LIN {X 0,Y 353.763,Z 539.719,A -85,B 0,C 180,E1 -13406.585,E2 -13406.585} C_VEL
LIN {X 0,Y 353.878,Z 540.945,A -85,B 0,C 180,E1 -13408.863,E2 -13408.863} C_VEL
LIN {X 0,Y 353.87,Z 540.944,A -85,B 0,C 180,E1 -13411.139,E2 -13411.139} C_VEL
LIN {X 0,Y 353.763,Z 539.714,A -85,B 0,C 180,E1 -13413.418,E2 -13413.418} C_VEL
LIN {X 0,Y 353.653,Z 537.275,A -85,B 0,C 180,E1 -13415.704,E2 -13415.704} C_VEL
LIN {X 0,Y 353.599,Z 534.658,A -85,B 0,C 180,E1 -13417.424,E2 -13417.424} C_VEL
LIN {X 0,Y 353.603,Z 529.946,A -85,B 0,C 180,E1 -13419.728,E2 -13419.728} C_VEL
LIN {X 0,Y 353.94,Z 523.835,A -85,B 0,C 180,E1 -13422.035,E2 -13422.035} C_VEL
LIN {X 0,Y 354.657,Z 516.159,A -85,B 0,C 180,E1 -13424.343,E2 -13424.343} C_VEL
LIN {X 0,Y 355.631,Z 507.936,A -85,B 0,C 180,E1 -13426.358,E2 -13426.358} C_VEL
LIN {X 0,Y 357.037,Z 498.093,A -85,B 0,C 180,E1 -13428.359,E2 -13428.359} C_VEL
LIN {X 0,Y 358.396,Z 488.39,A -85,B 0,C 180,E1 -13430.012,E2 -13430.012} C_VEL
LIN {X 0,Y 360.06,Z 477.162,A -85,B 0,C 180,E1 -13431.62,E2 -13431.62} C_VEL
LIN {X 0,Y 362.009,Z 464.197,A -85,B 0,C 180,E1 -13433.151,E2 -13433.151} C_VEL
LIN {X 0,Y 363.932,Z 451.379,A -85,B 0,C 180,E1 -13434.381,E2 -13434.381} C_VEL
LIN {X 0,Y 365.533,Z 438.976,A -85,B 0,C 180,E1 -13435.357,E2 -13435.357} C_VEL
LIN {X 0,Y 367.058,Z 425.471,A -85,B 0,C 180,E1 -13436.206,E2 -13436.206} C_VEL
LIN {X 0,Y 368.534,Z 409.817,A -85,B 0,C 180,E1 -13436.932,E2 -13436.932} C_VEL
LIN {X 0,Y 370.623,Z 388.777,A -85,B 0,C 180,E1 -13437.8,E2 -13437.8} C_VEL
LIN {X 0,Y 376.251,Z 305.9,A -85,B 0,C 180,E1 -13440.211,E2 -13440.211} C_VEL
LIN {X 0,Y 378.725,Z 273.446,A -85,B 0,C 180,E1 -13441.214,E2 -13441.214} C_VEL
LIN {X 0,Y 378.077,Z 256.965,A -85,B 0,C 180,E1 -13442.054,E2 -13442.054} C_VEL
LIN {X 0,Y 376.586,Z 241.39,A -85,B 0,C 180,E1 -13443.049,E2 -13443.049} C_VEL
LIN {X 0,Y 375.207,Z 230.072,A -85,B 0,C 180,E1 -13443.907,E2 -13443.907} C_VEL
LIN {X 0,Y 378.638,Z 218.88,A -85,B 0,C 180,E1 -13445.782,E2 -13445.782} C_VEL
LIN {X 0,Y 378.745,Z 217.493,A -85,B 0,C 180,E1 -13446.098,E2 -13446.098} C_VEL
LIN {X 0,Y 377.491,Z 211.701,A -85,B 0,C 180,E1 -13447.908,E2 -13447.908} C_VEL
LIN {X 0,Y 376.04,Z 206.391,A -85,B 0,C 180,E1 -13449.98,E2 -13449.98} C_VEL
LIN {X 0,Y 375.126,Z 203.374,A -85,B 0,C 180,E1 -13451.462,E2 -13451.462} C_VEL
LIN {X 0,Y 374.284,Z 201.061,A -85,B 0,C 180,E1 -13452.92,E2 -13452.92} C_VEL
LIN {X 0,Y 373.576,Z 199.328,A -85,B 0,C 180,E1 -13454.366,E2 -13454.366} C_VEL
LIN {X 0,Y 373.021,Z 198.122,A -85,B 0,C 180,E1 -13455.805,E2 -13455.805} C_VEL
LIN {X 0,Y 372.593,Z 197.372,A -85,B 0,C 180,E1 -13457.362,E2 -13457.362} C_VEL
LIN {X 0,Y 372.29,Z 197.213,A -85,B 0,C 180,E1 -13459.036,E2 -13459.036} C_VEL
LIN {X 0,Y 372.212,Z 198.099,A -85,B 0,C 180,E1 -13461.457,E2 -13461.457} C_VEL
LIN {X 0,Y 372.419,Z 199.091,A -85,B 0,C 180,E1 -13462.852,E2 -13462.852} C_VEL
LIN {X 0,Y 372.909,Z 202.358,A -85,B 0,C 180,E1 -13465.571,E2 -13465.571} C_VEL
LIN {X 0,Y 373.514,Z 206.249,A -85,B 0,C 180,E1 -13467.858,E2 -13467.858} C_VEL
LIN {X 0,Y 374.131,Z 211.79,A -85,B 0,C 180,E1 -13470.359,E2 -13470.359} C_VEL
LIN {X 0,Y 374.358,Z 214.356,A -85,B 0,C 180,E1 -13471.322,E2 -13471.322} C_VEL
LIN {X 0,Y 376.048,Z 218.405,A -85,B 0,C 180,E1 -13471.947,E2 -13471.947} C_VEL
LIN {X 0,Y 379.156,Z 231.614,A -85,B 0,C 180,E1 -13473.357,E2 -13473.357} C_VEL
LIN {X 0,Y 380.829,Z 240.437,A -85,B 0,C 180,E1 -13474.153,E2 -13474.153} C_VEL
LIN {X 0,Y 372.344,Z 323.117,A -85,B 0,C 180,E1 -13477.236,E2 -13477.236} C_VEL
LIN {X 0,Y 371.105,Z 340.845,A -85,B 0,C 180,E1 -13478.009,E2 -13478.009} C_VEL
LIN {X 0,Y 369.933,Z 354.657,A -85,B 0,C 180,E1 -13478.841,E2 -13478.841} C_VEL
LIN {X 0,Y 368.398,Z 368.573,A -85,B 0,C 180,E1 -13479.917,E2 -13479.917} C_VEL
LIN {X 0,Y 366.812,Z 380.901,A -85,B 0,C 180,E1 -13481.136,E2 -13481.136} C_VEL
LIN {X 0,Y 365.241,Z 392.111,A -85,B 0,C 180,E1 -13482.503,E2 -13482.503} C_VEL
LIN {X 0,Y 363.873,Z 400.494,A -85,B 0,C 180,E1 -13483.736,E2 -13483.736} C_VEL
LIN {X 0,Y 362.309,Z 409.709,A -85,B 0,C 180,E1 -13485.394,E2 -13485.394} C_VEL
LIN {X 0,Y 360.749,Z 417.376,A -85,B 0,C 180,E1 -13487.079,E2 -13487.079} C_VEL
LIN {X 0,Y 359.531,Z 423.347,A -85,B 0,C 180,E1 -13488.728,E2 -13488.728} C_VEL
LIN {X 0,Y 358.425,Z 428.175,A -85,B 0,C 180,E1 -13490.406,E2 -13490.406} C_VEL
LIN {X 0,Y 357.393,Z 431.88,A -85,B 0,C 180,E1 -13492.088,E2 -13492.088} C_VEL
LIN {X 0,Y 356.884,Z 433.766,A -85,B 0,C 180,E1 -13493.214,E2 -13493.214} C_VEL
LIN {X 0,Y 356.482,Z 435.152,A -85,B 0,C 180,E1 -13494.343,E2 -13494.343} C_VEL
LIN {X 0,Y 356.177,Z 436.114,A -85,B 0,C 180,E1 -13495.473,E2 -13495.473} C_VEL
LIN {X 0,Y 355.831,Z 436.688,A -85,B 0,C 180,E1 -13496.603,E2 -13496.603} C_VEL
LIN {X 0,Y 355.599,Z 436.836,A -85,B 0,C 180,E1 -13497.735,E2 -13497.735} C_VEL
LIN {X 0,Y 355.294,Z 436.541,A -85,B 0,C 180,E1 -13498.867,E2 -13498.867} C_VEL
LIN {X 0,Y 355.053,Z 435.824,A -85,B 0,C 180,E1 -13500,E2 -13500} C_VEL
LIN {X 0,Y 355.066,Z 434.672,A -85,B 0,C 180,E1 -13501.134,E2 -13501.134} C_VEL
LIN {X 0,Y 354.989,Z 432.145,A -85,B 0,C 180,E1 -13502.837,E2 -13502.837} C_VEL
LIN {X 0,Y 354.872,Z 428.61,A -85,B 0,C 180,E1 -13504.544,E2 -13504.544} C_VEL
LIN {X 0,Y 355.241,Z 423.954,A -85,B 0,C 180,E1 -13506.247,E2 -13506.247} C_VEL
LIN {X 0,Y 355.504,Z 418.114,A -85,B 0,C 180,E1 -13507.954,E2 -13507.954} C_VEL
LIN {X 0,Y 355.863,Z 410.905,A -85,B 0,C 180,E1 -13509.664,E2 -13509.664} C_VEL
LIN {X 0,Y 356.433,Z 402.004,A -85,B 0,C 180,E1 -13511.372,E2 -13511.372} C_VEL
LIN {X 0,Y 357.108,Z 391.08,A -85,B 0,C 180,E1 -13513.081,E2 -13513.081} C_VEL
LIN {X 0,Y 357.776,Z 379.778,A -85,B 0,C 180,E1 -13514.505,E2 -13514.505} C_VEL
LIN {X 0,Y 358.472,Z 367.292,A -85,B 0,C 180,E1 -13515.785,E2 -13515.785} C_VEL
LIN {X 0,Y 359.034,Z 354.854,A -85,B 0,C 180,E1 -13516.803,E2 -13516.803} C_VEL
LIN {X 0,Y 359.607,Z 340.6,A -85,B 0,C 180,E1 -13517.707,E2 -13517.707} C_VEL
LIN {X 0,Y 359.969,Z 327.731,A -85,B 0,C 180,E1 -13518.313,E2 -13518.313} C_VEL
LIN {X 0,Y 360.423,Z 308.207,A -85,B 0,C 180,E1 -13518.916,E2 -13518.916} C_VEL
LIN {X 0,Y 362.911,Z 226.278,A -85,B 0,C 180,E1 -13521.162,E2 -13521.162} C_VEL
LIN {X 0,Y 359.275,Z 202.978,A -85,B 0,C 180,E1 -13522.026,E2 -13522.026} C_VEL
LIN {X 0,Y 360.736,Z 186.431,A -85,B 0,C 180,E1 -13525.38,E2 -13525.38} C_VEL
LIN {X 0,Y 360.386,Z 182.557,A -85,B 0,C 180,E1 -13526.224,E2 -13526.224} C_VEL
LIN {X 0,Y 357.643,Z 170.027,A -85,B 0,C 180,E1 -13529.101,E2 -13529.101} C_VEL
LIN {X 0,Y 354.837,Z 157.912,A -85,B 0,C 180,E1 -13532.024,E2 -13532.024} C_VEL
LIN {X 0,Y 354.827,Z 157.912,A -85,B 0,C 180,E1 -13535.699,E2 -13535.699} C_VEL
LIN {X 0,Y 354.804,Z 157.904,A -85,B 0,C 180,E1 -13539.418,E2 -13539.418} C_VEL
LIN {X 0,Y 354.791,Z 157.912,A -85,B 0,C 180,E1 -13542.866,E2 -13542.866} C_VEL
LIN {X 0,Y 354.786,Z 157.915,A -85,B 0,C 180,E1 -13546.105,E2 -13546.105} C_VEL
LIN {X 0,Y 354.793,Z 157.914,A -85,B 0,C 180,E1 -13549.178,E2 -13549.178} C_VEL
LIN {X 0,Y 354.812,Z 157.912,A -85,B 0,C 180,E1 -13552.402,E2 -13552.402} C_VEL
LIN {X 0,Y 354.888,Z 158.025,A -85,B 0,C 180,E1 -13555.059,E2 -13555.059} C_VEL
LIN {X 0,Y 359.7,Z 171.926,A -85,B 0,C 180,E1 -13557.692,E2 -13557.692} C_VEL
LIN {X 0,Y 369.684,Z 191.582,A -85,B 0,C 180,E1 -13559.124,E2 -13559.124} C_VEL
LIN {X 0,Y 374.764,Z 202.976,A -85,B 0,C 180,E1 -13559.846,E2 -13559.846} C_VEL
LIN {X 0,Y 372.675,Z 285.003,A -85,B 0,C 180,E1 -13561.448,E2 -13561.448} C_VEL
LIN {X 0,Y 371.249,Z 338.669,A -85,B 0,C 180,E1 -13562.519,E2 -13562.519} C_VEL
LIN {X 0,Y 370.646,Z 353.596,A -85,B 0,C 180,E1 -13563.016,E2 -13563.016} C_VEL
LIN {X 0,Y 369.847,Z 366.135,A -85,B 0,C 180,E1 -13563.599,E2 -13563.599} C_VEL
LIN {X 0,Y 368.737,Z 380.111,A -85,B 0,C 180,E1 -13564.453,E2 -13564.453} C_VEL
LIN {X 0,Y 367.253,Z 394.224,A -85,B 0,C 180,E1 -13565.553,E2 -13565.553} C_VEL
LIN {X 0,Y 365.586,Z 407.061,A -85,B 0,C 180,E1 -13566.789,E2 -13566.789} C_VEL
LIN {X 0,Y 363.719,Z 419.822,A -85,B 0,C 180,E1 -13568.297,E2 -13568.297} C_VEL
LIN {X 0,Y 362.183,Z 430.662,A -85,B 0,C 180,E1 -13569.852,E2 -13569.852} C_VEL
LIN {X 0,Y 360.499,Z 440.551,A -85,B 0,C 180,E1 -13571.529,E2 -13571.529} C_VEL
LIN {X 0,Y 358.745,Z 450.446,A -85,B 0,C 180,E1 -13573.554,E2 -13573.554} C_VEL
LIN {X 0,Y 357.303,Z 459.202,A -85,B 0,C 180,E1 -13575.765,E2 -13575.765} C_VEL
LIN {X 0,Y 356.039,Z 466.459,A -85,B 0,C 180,E1 -13578.037,E2 -13578.037} C_VEL
LIN {X 0,Y 355.175,Z 472.199,A -85,B 0,C 180,E1 -13580.316,E2 -13580.316} C_VEL
LIN {X 0,Y 354.597,Z 476.084,A -85,B 0,C 180,E1 -13582.302,E2 -13582.302} C_VEL
LIN {X 0,Y 354.189,Z 479.036,A -85,B 0,C 180,E1 -13584.305,E2 -13584.305} C_VEL
LIN {X 0,Y 353.991,Z 481.303,A -85,B 0,C 180,E1 -13586.584,E2 -13586.584} C_VEL
LIN {X 0,Y 353.777,Z 482.464,A -85,B 0,C 180,E1 -13588.86,E2 -13588.86} C_VEL
LIN {X 0,Y 353.777,Z 482.478,A -85,B 0,C 180,E1 -13591.137,E2 -13591.137} C_VEL
LIN {X 0,Y 353.85,Z 482.051,A -85,B 0,C 180,E1 -13592.295,E2 -13592.295} C_VEL
LIN {X 0,Y 353.242,Z 481.561,A -85,B 0,C 180,E1 -13593.242,E2 -13593.242} C_VEL
LIN {X 0,Y 350.492,Z 480.531,A -85,B 0,C 180,E1 -13594.786,E2 -13594.786} C_VEL
LIN {X 0,Y 348.245,Z 479.373,A -85,B 0,C 180,E1 -13596.027,E2 -13596.027} C_VEL
LIN {X 0,Y 347.422,Z 478.194,A -85,B 0,C 180,E1 -13596.975,E2 -13596.975} C_VEL
LIN {X 0,Y 347.431,Z 477.716,A -85,B 0,C 180,E1 -13597.292,E2 -13597.292} C_VEL
LIN {X 0,Y 347.976,Z 474.204,A -85,B 0,C 180,E1 -13599.297,E2 -13599.297} C_VEL
LIN {X 0,Y 348.813,Z 468.885,A -85,B 0,C 180,E1 -13601.622,E2 -13601.622} C_VEL
LIN {X 0,Y 349.961,Z 462.092,A -85,B 0,C 180,E1 -13603.943,E2 -13603.943} C_VEL
LIN {X 0,Y 351.287,Z 454.677,A -85,B 0,C 180,E1 -13605.997,E2 -13605.997} C_VEL
LIN {X 0,Y 352.908,Z 445.996,A -85,B 0,C 180,E1 -13607.978,E2 -13607.978} C_VEL
LIN {X 0,Y 354.83,Z 435.328,A -85,B 0,C 180,E1 -13609.977,E2 -13609.977} C_VEL
LIN {X 0,Y 356.6,Z 424.361,A -85,B 0,C 180,E1 -13611.685,E2 -13611.685} C_VEL
LIN {X 0,Y 358.482,Z 412.292,A -85,B 0,C 180,E1 -13613.236,E2 -13613.236} C_VEL
LIN {X 0,Y 360.37,Z 398.941,A -85,B 0,C 180,E1 -13614.635,E2 -13614.635} C_VEL
LIN {X 0,Y 361.89,Z 385.861,A -85,B 0,C 180,E1 -13615.753,E2 -13615.753} C_VEL
LIN {X 0,Y 363.247,Z 372.108,A -85,B 0,C 180,E1 -13616.688,E2 -13616.688} C_VEL
LIN {X 0,Y 364.171,Z 357.951,A -85,B 0,C 180,E1 -13617.438,E2 -13617.438} C_VEL
LIN {X 0,Y 364.941,Z 342.964,A -85,B 0,C 180,E1 -13617.994,E2 -13617.994} C_VEL
LIN {X 0,Y 365.469,Z 322.552,A -85,B 0,C 180,E1 -13618.458,E2 -13618.458} C_VEL
LIN {X 0,Y 368.091,Z 226.756,A -85,B 0,C 180,E1 -13620.348,E2 -13620.348} C_VEL
LIN {X 0,Y 368.573,Z 204.816,A -85,B 0,C 180,E1 -13620.794,E2 -13620.794} C_VEL
LIN {X 0,Y 361.129,Z 188.738,A -85,B 0,C 180,E1 -13621.884,E2 -13621.884} C_VEL
LIN {X 0,Y 352.618,Z 172.366,A -85,B 0,C 180,E1 -13623.165,E2 -13623.165} C_VEL
LIN {X 0,Y 347.762,Z 158.793,A -85,B 0,C 180,E1 -13625.847,E2 -13625.847} C_VEL
LIN {X 0,Y 347.747,Z 158.778,A -85,B 0,C 180,E1 -13628.791,E2 -13628.791} C_VEL
LIN {X 0,Y 347.748,Z 158.783,A -85,B 0,C 180,E1 -13631.828,E2 -13631.828} C_VEL
LIN {X 0,Y 347.727,Z 158.79,A -85,B 0,C 180,E1 -13635.021,E2 -13635.021} C_VEL
LIN {X 0,Y 347.761,Z 158.787,A -85,B 0,C 180,E1 -13638.393,E2 -13638.393} C_VEL
LIN {X 0,Y 347.768,Z 158.785,A -85,B 0,C 180,E1 -13642.009,E2 -13642.009} C_VEL
LIN {X 0,Y 347.736,Z 158.783,A -85,B 0,C 180,E1 -13645.535,E2 -13645.535} C_VEL
LIN {X 0,Y 347.756,Z 158.791,A -85,B 0,C 180,E1 -13648.301,E2 -13648.301} C_VEL
LIN {X 0,Y 347.797,Z 158.775,A -85,B 0,C 180,E1 -13650.989,E2 -13650.989} C_VEL
LIN {X 0,Y 347.822,Z 158.779,A -85,B 0,C 180,E1 -13653.607,E2 -13653.607} C_VEL
LIN {X 0,Y 347.775,Z 158.779,A -85,B 0,C 180,E1 -13656.161,E2 -13656.161} C_VEL
LIN {X 0,Y 347.801,Z 158.776,A -85,B 0,C 180,E1 -13659.909,E2 -13659.909} C_VEL
LIN {X 0,Y 347.856,Z 158.77,A -85,B 0,C 180,E1 -13662.359,E2 -13662.359} C_VEL
LIN {X 0,Y 347.887,Z 158.765,A -85,B 0,C 180,E1 -13665.97,E2 -13665.97} C_VEL
LIN {X 0,Y 347.918,Z 158.771,A -85,B 0,C 180,E1 -13669.525,E2 -13669.525} C_VEL
LIN {X 0,Y 348.063,Z 158.747,A -85,B 0,C 180,E1 -13671.874,E2 -13671.874} C_VEL
LIN {X 0,Y 348.057,Z 158.734,A -85,B 0,C 180,E1 -13674.205,E2 -13674.205} C_VEL
LIN {X 0,Y 348.198,Z 158.734,A -85,B 0,C 180,E1 -13677.686,E2 -13677.686} C_VEL
LIN {X 0,Y 348.358,Z 158.695,A -85,B 0,C 180,E1 -13680,E2 -13680} C_VEL
LIN {X 0,Y 348.198,Z 158.73,A -85,B 0,C 180,E1 -13682.313,E2 -13682.313} C_VEL
LIN {X 0,Y 348.095,Z 158.727,A -85,B 0,C 180,E1 -13686.958,E2 -13686.958} C_VEL
LIN {X 0,Y 347.956,Z 158.762,A -85,B 0,C 180,E1 -13689.299,E2 -13689.299} C_VEL
LIN {X 0,Y 347.879,Z 158.753,A -85,B 0,C 180,E1 -13692.84,E2 -13692.84} C_VEL
LIN {X 0,Y 347.83,Z 158.78,A -85,B 0,C 180,E1 -13696.432,E2 -13696.432} C_VEL
LIN {X 0,Y 347.84,Z 158.761,A -85,B 0,C 180,E1 -13698.861,E2 -13698.861} C_VEL
LIN {X 0,Y 347.764,Z 158.786,A -85,B 0,C 180,E1 -13702.58,E2 -13702.58} C_VEL
LIN {X 0,Y 347.801,Z 158.772,A -85,B 0,C 180,E1 -13705.109,E2 -13705.109} C_VEL
LIN {X 0,Y 347.798,Z 158.786,A -85,B 0,C 180,E1 -13707.695,E2 -13707.695} C_VEL
LIN {X 0,Y 347.739,Z 158.783,A -85,B 0,C 180,E1 -13710.349,E2 -13710.349} C_VEL
LIN {X 0,Y 347.738,Z 158.784,A -85,B 0,C 180,E1 -13714.045,E2 -13714.045} C_VEL
LIN {X 0,Y 347.757,Z 158.79,A -85,B 0,C 180,E1 -13717.321,E2 -13717.321} C_VEL
LIN {X 0,Y 347.722,Z 158.752,A -85,B 0,C 180,E1 -13720.298,E2 -13720.298} C_VEL
LIN {X 0,Y 347.72,Z 158.795,A -85,B 0,C 180,E1 -13723.408,E2 -13723.408} C_VEL
LIN {X 0,Y 347.778,Z 158.79,A -85,B 0,C 180,E1 -13726.677,E2 -13726.677} C_VEL
LIN {X 0,Y 347.827,Z 158.983,A -85,B 0,C 180,E1 -13728.726,E2 -13728.726} C_VEL
LIN {X 0,Y 353.697,Z 178.827,A -85,B 0,C 180,E1 -13732.395,E2 -13732.395} C_VEL
LIN {X 0,Y 359.113,Z 197.549,A -85,B 0,C 180,E1 -13735.625,E2 -13735.625} C_VEL
LIN {X 0,Y 360.254,Z 202.214,A -85,B 0,C 180,E1 -13736.391,E2 -13736.391} C_VEL
LIN {X 0,Y 359.364,Z 209.237,A -85,B 0,C 180,E1 -13737.323,E2 -13737.323} C_VEL
LIN {X 0,Y 360.134,Z 219.316,A -85,B 0,C 180,E1 -13737.839,E2 -13737.839} C_VEL
LIN {X 0,Y 365.985,Z 269.667,A -85,B 0,C 180,E1 -13739.525,E2 -13739.525} C_VEL
LIN {X 0,Y 366.395,Z 275.472,A -85,B 0,C 180,E1 -13739.69,E2 -13739.69} C_VEL
LIN {X 0,Y 363.207,Z 392.946,A -85,B 0,C 180,E1 -13742.017,E2 -13742.017} C_VEL
LIN {X 0,Y 362.288,Z 407.953,A -85,B 0,C 180,E1 -13742.49,E2 -13742.49} C_VEL
LIN {X 0,Y 360.903,Z 422.665,A -85,B 0,C 180,E1 -13743.159,E2 -13743.159} C_VEL
LIN {X 0,Y 359.199,Z 437.235,A -85,B 0,C 180,E1 -13744.055,E2 -13744.055} C_VEL
LIN {X 0,Y 357.445,Z 451.111,A -85,B 0,C 180,E1 -13745.161,E2 -13745.161} C_VEL
LIN {X 0,Y 355.396,Z 463.777,A -85,B 0,C 180,E1 -13746.396,E2 -13746.396} C_VEL
LIN {X 0,Y 353.42,Z 476.713,A -85,B 0,C 180,E1 -13747.956,E2 -13747.956} C_VEL
LIN {X 0,Y 351.695,Z 487.545,A -85,B 0,C 180,E1 -13749.532,E2 -13749.532} C_VEL
LIN {X 0,Y 350.176,Z 497.585,A -85,B 0,C 180,E1 -13751.271,E2 -13751.271} C_VEL
LIN {X 0,Y 348.867,Z 506.148,A -85,B 0,C 180,E1 -13753.018,E2 -13753.018} C_VEL
LIN {X 0,Y 347.793,Z 514.543,A -85,B 0,C 180,E1 -13755.071,E2 -13755.071} C_VEL
LIN {X 0,Y 347.028,Z 521.509,A -85,B 0,C 180,E1 -13757.13,E2 -13757.13} C_VEL
LIN {X 0,Y 346.539,Z 527.985,A -85,B 0,C 180,E1 -13759.485,E2 -13759.485} C_VEL
LIN {X 0,Y 346.461,Z 533.011,A -85,B 0,C 180,E1 -13761.838,E2 -13761.838} C_VEL
LIN {X 0,Y 346.563,Z 536.701,A -85,B 0,C 180,E1 -13764.182,E2 -13764.182} C_VEL
LIN {X 0,Y 346.665,Z 539.132,A -85,B 0,C 180,E1 -13766.515,E2 -13766.515} C_VEL
LIN {X 0,Y 346.824,Z 540.362,A -85,B 0,C 180,E1 -13768.84,E2 -13768.84} C_VEL
LIN {X 0,Y 346.817,Z 540.361,A -85,B 0,C 180,E1 -13771.163,E2 -13771.163} C_VEL
LIN {X 0,Y 346.665,Z 539.126,A -85,B 0,C 180,E1 -13773.488,E2 -13773.488} C_VEL
LIN {X 0,Y 346.582,Z 536.688,A -85,B 0,C 180,E1 -13775.821,E2 -13775.821} C_VEL
LIN {X 0,Y 346.479,Z 532.983,A -85,B 0,C 180,E1 -13778.164,E2 -13778.164} C_VEL
LIN {X 0,Y 346.578,Z 527.946,A -85,B 0,C 180,E1 -13780.517,E2 -13780.517} C_VEL
LIN {X 0,Y 347.068,Z 521.466,A -85,B 0,C 180,E1 -13782.872,E2 -13782.872} C_VEL
LIN {X 0,Y 347.81,Z 514.488,A -85,B 0,C 180,E1 -13784.931,E2 -13784.931} C_VEL
LIN {X 0,Y 348.919,Z 506.079,A -85,B 0,C 180,E1 -13786.983,E2 -13786.983} C_VEL
LIN {X 0,Y 350.429,Z 496.148,A -85,B 0,C 180,E1 -13788.988,E2 -13788.988} C_VEL
LIN {X 0,Y 351.991,Z 485.637,A -85,B 0,C 180,E1 -13790.758,E2 -13790.758} C_VEL
LIN {X 0,Y 353.965,Z 473.341,A -85,B 0,C 180,E1 -13792.472,E2 -13792.472} C_VEL
LIN {X 0,Y 356.088,Z 459.655,A -85,B 0,C 180,E1 -13794.022,E2 -13794.022} C_VEL
LIN {X 0,Y 358.062,Z 445.95,A -85,B 0,C 180,E1 -13795.273,E2 -13795.273} C_VEL
LIN {X 0,Y 359.886,Z 431.721,A -85,B 0,C 180,E1 -13796.3,E2 -13796.3} C_VEL
LIN {X 0,Y 361.501,Z 417.029,A -85,B 0,C 180,E1 -13797.108,E2 -13797.108} C_VEL
LIN {X 0,Y 363.932,Z 398.14,A -85,B 0,C 180,E1 -13798.082,E2 -13798.082} C_VEL
LIN {X 0,Y 365.464,Z 381.659,A -85,B 0,C 180,E1 -13798.697,E2 -13798.697} C_VEL
LIN {X 0,Y 370.169,Z 317.229,A -85,B 0,C 180,E1 -13800.603,E2 -13800.603} C_VEL
LIN {X 0,Y 373.714,Z 274.991,A -85,B 0,C 180,E1 -13801.938,E2 -13801.938} C_VEL
LIN {X 0,Y 373.221,Z 259.069,A -85,B 0,C 180,E1 -13802.777,E2 -13802.777} C_VEL
LIN {X 0,Y 371.973,Z 243.743,A -85,B 0,C 180,E1 -13803.791,E2 -13803.791} C_VEL
LIN {X 0,Y 370.399,Z 229.425,A -85,B 0,C 180,E1 -13804.945,E2 -13804.945} C_VEL
LIN {X 0,Y 373.015,Z 221.289,A -85,B 0,C 180,E1 -13806.381,E2 -13806.381} C_VEL
LIN {X 0,Y 371.827,Z 215.544,A -85,B 0,C 180,E1 -13808.241,E2 -13808.241} C_VEL
LIN {X 0,Y 370.359,Z 209.828,A -85,B 0,C 180,E1 -13810.62,E2 -13810.62} C_VEL
LIN {X 0,Y 369.48,Z 207.102,A -85,B 0,C 180,E1 -13812.112,E2 -13812.112} C_VEL
LIN {X 0,Y 368.695,Z 205.03,A -85,B 0,C 180,E1 -13813.585,E2 -13813.585} C_VEL
LIN {X 0,Y 368.052,Z 203.519,A -85,B 0,C 180,E1 -13815.048,E2 -13815.048} C_VEL
LIN {X 0,Y 367.52,Z 202.469,A -85,B 0,C 180,E1 -13816.609,E2 -13816.609} C_VEL
LIN {X 0,Y 367.155,Z 201.985,A -85,B 0,C 180,E1 -13818.292,E2 -13818.292} C_VEL
LIN {X 0,Y 366.898,Z 202.44,A -85,B 0,C 180,E1 -13820.793,E2 -13820.793} C_VEL
LIN {X 0,Y 366.958,Z 203.261,A -85,B 0,C 180,E1 -13822.203,E2 -13822.203} C_VEL
LIN {X 0,Y 367.3,Z 206.132,A -85,B 0,C 180,E1 -13824.969,E2 -13824.969} C_VEL
LIN {X 0,Y 367.772,Z 209.601,A -85,B 0,C 180,E1 -13827.229,E2 -13827.229} C_VEL
LIN {X 0,Y 368.272,Z 214.827,A -85,B 0,C 180,E1 -13829.773,E2 -13829.773} C_VEL
LIN {X 0,Y 368.538,Z 215.694,A -85,B 0,C 180,E1 -13830.04,E2 -13830.04} C_VEL
LIN {X 0,Y 371.209,Z 220.927,A -85,B 0,C 180,E1 -13831.065,E2 -13831.065} C_VEL
LIN {X 0,Y 372.143,Z 223.669,A -85,B 0,C 180,E1 -13831.464,E2 -13831.464} C_VEL
LIN {X 0,Y 374.899,Z 236.499,A -85,B 0,C 180,E1 -13832.858,E2 -13832.858} C_VEL
LIN {X 0,Y 375.941,Z 242.696,A -85,B 0,C 180,E1 -13833.428,E2 -13833.428} C_VEL
LIN {X 0,Y 366.955,Z 323.86,A -85,B 0,C 180,E1 -13836.532,E2 -13836.532} C_VEL
LIN {X 0,Y 365.598,Z 341.651,A -85,B 0,C 180,E1 -13837.329,E2 -13837.329} C_VEL
LIN {X 0,Y 364.363,Z 354.916,A -85,B 0,C 180,E1 -13838.134,E2 -13838.134} C_VEL
LIN {X 0,Y 362.669,Z 369.199,A -85,B 0,C 180,E1 -13839.252,E2 -13839.252} C_VEL
LIN {X 0,Y 360.919,Z 381.86,A -85,B 0,C 180,E1 -13840.521,E2 -13840.521} C_VEL
LIN {X 0,Y 359.214,Z 393.033,A -85,B 0,C 180,E1 -13841.905,E2 -13841.905} C_VEL
LIN {X 0,Y 357.737,Z 401.41,A -85,B 0,C 180,E1 -13843.156,E2 -13843.156} C_VEL
LIN {X 0,Y 356.051,Z 410.649,A -85,B 0,C 180,E1 -13844.839,E2 -13844.839} C_VEL
LIN {X 0,Y 354.316,Z 418.652,A -85,B 0,C 180,E1 -13846.632,E2 -13846.632} C_VEL
LIN {X 0,Y 352.819,Z 425.248,A -85,B 0,C 180,E1 -13848.51,E2 -13848.51} C_VEL
LIN {X 0,Y 351.647,Z 429.9,A -85,B 0,C 180,E1 -13850.219,E2 -13850.219} C_VEL
LIN {X 0,Y 350.561,Z 433.461,A -85,B 0,C 180,E1 -13851.933,E2 -13851.933} C_VEL
LIN {X 0,Y 349.99,Z 435.223,A -85,B 0,C 180,E1 -13853.08,E2 -13853.08} C_VEL
LIN {X 0,Y 349.568,Z 436.525,A -85,B 0,C 180,E1 -13854.231,E2 -13854.231} C_VEL
LIN {X 0,Y 349.221,Z 437.423,A -85,B 0,C 180,E1 -13855.383,E2 -13855.383} C_VEL
LIN {X 0,Y 348.858,Z 437.921,A -85,B 0,C 180,E1 -13856.535,E2 -13856.535} C_VEL
LIN {X 0,Y 348.608,Z 437.957,A -85,B 0,C 180,E1 -13857.689,E2 -13857.689} C_VEL
LIN {X 0,Y 348.285,Z 437.584,A -85,B 0,C 180,E1 -13858.844,E2 -13858.844} C_VEL
LIN {X 0,Y 348.026,Z 436.798,A -85,B 0,C 180,E1 -13860,E2 -13860} C_VEL
LIN {X 0,Y 348.04,Z 435.574,A -85,B 0,C 180,E1 -13861.157,E2 -13861.157} C_VEL
LIN {X 0,Y 347.951,Z 432.916,A -85,B 0,C 180,E1 -13862.895,E2 -13862.895} C_VEL
LIN {X 0,Y 347.844,Z 429.246,A -85,B 0,C 180,E1 -13864.636,E2 -13864.636} C_VEL
LIN {X 0,Y 348.201,Z 424.451,A -85,B 0,C 180,E1 -13866.374,E2 -13866.374} C_VEL
LIN {X 0,Y 348.477,Z 418.463,A -85,B 0,C 180,E1 -13868.116,E2 -13868.116} C_VEL
LIN {X 0,Y 348.85,Z 411.051,A -85,B 0,C 180,E1 -13869.86,E2 -13869.86} C_VEL
LIN {X 0,Y 349.437,Z 401.938,A -85,B 0,C 180,E1 -13871.603,E2 -13871.603} C_VEL
LIN {X 0,Y 350.09,Z 391.773,A -85,B 0,C 180,E1 -13873.2,E2 -13873.2} C_VEL
LIN {X 0,Y 350.778,Z 380.414,A -85,B 0,C 180,E1 -13874.652,E2 -13874.652} C_VEL
LIN {X 0,Y 351.479,Z 367.878,A -85,B 0,C 180,E1 -13875.958,E2 -13875.958} C_VEL
LIN {X 0,Y 352.078,Z 355.174,A -85,B 0,C 180,E1 -13877.011,E2 -13877.011} C_VEL
LIN {X 0,Y 352.657,Z 341.115,A -85,B 0,C 180,E1 -13877.918,E2 -13877.918} C_VEL
LIN {X 0,Y 353.037,Z 328.228,A -85,B 0,C 180,E1 -13878.536,E2 -13878.536} C_VEL
LIN {X 0,Y 353.519,Z 307.596,A -85,B 0,C 180,E1 -13879.187,E2 -13879.187} C_VEL
LIN {X 0,Y 356.105,Z 227.175,A -85,B 0,C 180,E1 -13881.45,E2 -13881.45} C_VEL
LIN {X 0,Y 352.399,Z 203.154,A -85,B 0,C 180,E1 -13882.383,E2 -13882.383} C_VEL
LIN {X 0,Y 353.845,Z 187.528,A -85,B 0,C 180,E1 -13885.594,E2 -13885.594} C_VEL
LIN {X 0,Y 353.382,Z 183.465,A -85,B 0,C 180,E1 -13886.496,E2 -13886.496} C_VEL
LIN {X 0,Y 350.612,Z 171,A -85,B 0,C 180,E1 -13889.413,E2 -13889.413} C_VEL
LIN {X 0,Y 347.772,Z 158.791,A -85,B 0,C 180,E1 -13892.373,E2 -13892.373} C_VEL
LIN {X 0,Y 347.775,Z 158.79,A -85,B 0,C 180,E1 -13896.064,E2 -13896.064} C_VEL
LIN {X 0,Y 347.737,Z 158.79,A -85,B 0,C 180,E1 -13898.795,E2 -13898.795} C_VEL
LIN {X 0,Y 347.753,Z 158.793,A -85,B 0,C 180,E1 -13901.83,E2 -13901.83} C_VEL
LIN {X 0,Y 347.772,Z 158.788,A -85,B 0,C 180,E1 -13905.016,E2 -13905.016} C_VEL
LIN {X 0,Y 347.756,Z 158.793,A -85,B 0,C 180,E1 -13908.396,E2 -13908.396} C_VEL
LIN {X 0,Y 347.778,Z 158.791,A -85,B 0,C 180,E1 -13912.011,E2 -13912.011} C_VEL
LIN {X 0,Y 347.786,Z 158.793,A -85,B 0,C 180,E1 -13914.298,E2 -13914.298} C_VEL
LIN {X 0,Y 352.675,Z 172.62,A -85,B 0,C 180,E1 -13916.97,E2 -13916.97} C_VEL
LIN {X 0,Y 362.527,Z 191.569,A -85,B 0,C 180,E1 -13918.431,E2 -13918.431} C_VEL
LIN {X 0,Y 368.636,Z 204.951,A -85,B 0,C 180,E1 -13919.324,E2 -13919.324} C_VEL
LIN {X 0,Y 366.448,Z 285.768,A -85,B 0,C 180,E1 -13920.923,E2 -13920.923} C_VEL
LIN {X 0,Y 364.942,Z 340.552,A -85,B 0,C 180,E1 -13922.042,E2 -13922.042} C_VEL
LIN {X 0,Y 364.238,Z 355.662,A -85,B 0,C 180,E1 -13922.57,E2 -13922.57} C_VEL
LIN {X 0,Y 363.324,Z 370.003,A -85,B 0,C 180,E1 -13923.294,E2 -13923.294} C_VEL
LIN {X 0,Y 362.204,Z 382.587,A -85,B 0,C 180,E1 -13924.113,E2 -13924.113} C_VEL
LIN {X 0,Y 360.652,Z 396.322,A -85,B 0,C 180,E1 -13925.229,E2 -13925.229} C_VEL
LIN {X 0,Y 358.709,Z 410.137,A -85,B 0,C 180,E1 -13926.624,E2 -13926.624} C_VEL
LIN {X 0,Y 356.808,Z 422.574,A -85,B 0,C 180,E1 -13928.173,E2 -13928.173} C_VEL
LIN {X 0,Y 355.232,Z 432.971,A -85,B 0,C 180,E1 -13929.742,E2 -13929.742} C_VEL
LIN {X 0,Y 353.513,Z 442.593,A -85,B 0,C 180,E1 -13931.451,E2 -13931.451} C_VEL
LIN {X 0,Y 351.962,Z 451.03,A -85,B 0,C 180,E1 -13933.228,E2 -13933.228} C_VEL
LIN {X 0,Y 350.443,Z 459.787,A -85,B 0,C 180,E1 -13935.481,E2 -13935.481} C_VEL
LIN {X 0,Y 349.12,Z 467.044,A -85,B 0,C 180,E1 -13937.796,E2 -13937.796} C_VEL
LIN {X 0,Y 348.187,Z 472.785,A -85,B 0,C 180,E1 -13940.12,E2 -13940.12} C_VEL
LIN {X 0,Y 347.562,Z 476.822,A -85,B 0,C 180,E1 -13942.233,E2 -13942.233} C_VEL
LIN {X 0,Y 347.135,Z 479.622,A -85,B 0,C 180,E1 -13944.189,E2 -13944.189} C_VEL
LIN {X 0,Y 346.938,Z 481.887,A -85,B 0,C 180,E1 -13946.514,E2 -13946.514} C_VEL
LIN {X 0,Y 346.702,Z 483.049,A -85,B 0,C 180,E1 -13948.837,E2 -13948.837} C_VEL
LIN {X 0,Y 346.702,Z 483.063,A -85,B 0,C 180,E1 -13951.16,E2 -13951.16} C_VEL
LIN {X 0,Y 346.935,Z 481.954,A -85,B 0,C 180,E1 -13953.483,E2 -13953.483} C_VEL
LIN {X 0,Y 347.122,Z 479.747,A -85,B 0,C 180,E1 -13955.809,E2 -13955.809} C_VEL
LIN {X 0,Y 347.431,Z 477.716,A -85,B 0,C 180,E1 -13957.292,E2 -13957.292} C_VEL
LIN {X 0,Y 347.046,Z 476.273,A -85,B 0,C 180,E1 -13958.235,E2 -13958.235} C_VEL
LIN {X 0,Y 344.635,Z 473.732,A -85,B 0,C 180,E1 -13959.774,E2 -13959.774} C_VEL
LIN {X 0,Y 342.635,Z 471.38,A -85,B 0,C 180,E1 -13961,E2 -13961} C_VEL
LIN {X 0,Y 341.982,Z 469.302,A -85,B 0,C 180,E1 -13961.923,E2 -13961.923} C_VEL
LIN {X 0,Y 342.045,Z 468.505,A -85,B 0,C 180,E1 -13962.228,E2 -13962.228} C_VEL
LIN {X 0,Y 343.078,Z 462.675,A -85,B 0,C 180,E1 -13964.229,E2 -13964.229} C_VEL
LIN {X 0,Y 344.429,Z 455.517,A -85,B 0,C 180,E1 -13966.258,E2 -13966.258} C_VEL
LIN {X 0,Y 346.189,Z 446.574,A -85,B 0,C 180,E1 -13968.339,E2 -13968.339} C_VEL
LIN {X 0,Y 348.186,Z 435.903,A -85,B 0,C 180,E1 -13970.375,E2 -13970.375} C_VEL
LIN {X 0,Y 350.02,Z 424.936,A -85,B 0,C 180,E1 -13972.114,E2 -13972.114} C_VEL
LIN {X 0,Y 351.982,Z 412.862,A -85,B 0,C 180,E1 -13973.691,E2 -13973.691} C_VEL
LIN {X 0,Y 353.946,Z 399.506,A -85,B 0,C 180,E1 -13975.112,E2 -13975.112} C_VEL
LIN {X 0,Y 355.539,Z 386.417,A -85,B 0,C 180,E1 -13976.248,E2 -13976.248} C_VEL
LIN {X 0,Y 356.931,Z 372.786,A -85,B 0,C 180,E1 -13977.19,E2 -13977.19} C_VEL
LIN {X 0,Y 357.903,Z 358.645,A -85,B 0,C 180,E1 -13977.951,E2 -13977.951} C_VEL
LIN {X 0,Y 358.721,Z 343.466,A -85,B 0,C 180,E1 -13978.524,E2 -13978.524} C_VEL
LIN {X 0,Y 359.259,Z 323.001,A -85,B 0,C 180,E1 -13978.996,E2 -13978.996} C_VEL
LIN {X 0,Y 362.012,Z 227.212,A -85,B 0,C 180,E1 -13980.913,E2 -13980.913} C_VEL
LIN {X 0,Y 362.549,Z 207.084,A -85,B 0,C 180,E1 -13981.321,E2 -13981.321} C_VEL
LIN {X 0,Y 355.68,Z 192.227,A -85,B 0,C 180,E1 -13982.359,E2 -13982.359} C_VEL
LIN {X 0,Y 346.747,Z 175.208,A -85,B 0,C 180,E1 -13983.733,E2 -13983.733} C_VEL
LIN {X 0,Y 345.548,Z 172.887,A -85,B 0,C 180,E1 -13983.944,E2 -13983.944} C_VEL
LIN {X 0,Y 341.659,Z 162.406,A -85,B 0,C 180,E1 -13986.027,E2 -13986.027} C_VEL
LIN {X 0,Y 340.709,Z 159.667,A -85,B 0,C 180,E1 -13986.639,E2 -13986.639} C_VEL
LIN {X 0,Y 340.683,Z 159.645,A -85,B 0,C 180,E1 -13990.246,E2 -13990.246} C_VEL
LIN {X 0,Y 340.654,Z 159.67,A -85,B 0,C 180,E1 -13993.773,E2 -13993.773} C_VEL
LIN {X 0,Y 340.723,Z 159.661,A -85,B 0,C 180,E1 -13997.947,E2 -13997.947} C_VEL
LIN {X 0,Y 340.731,Z 159.659,A -85,B 0,C 180,E1 -14001.772,E2 -14001.772} C_VEL
LIN {X 0,Y 340.714,Z 159.658,A -85,B 0,C 180,E1 -14005.594,E2 -14005.594} C_VEL
LIN {X 0,Y 340.707,Z 159.661,A -85,B 0,C 180,E1 -14008.956,E2 -14008.956} C_VEL
LIN {X 0,Y 340.77,Z 159.662,A -85,B 0,C 180,E1 -14012.473,E2 -14012.473} C_VEL
LIN {X 0,Y 340.744,Z 159.65,A -85,B 0,C 180,E1 -14015.637,E2 -14015.637} C_VEL
LIN {X 0,Y 340.733,Z 159.658,A -85,B 0,C 180,E1 -14019.473,E2 -14019.473} C_VEL
LIN {X 0,Y 340.847,Z 159.641,A -85,B 0,C 180,E1 -14021.984,E2 -14021.984} C_VEL
LIN {X 0,Y 340.859,Z 159.642,A -85,B 0,C 180,E1 -14025.704,E2 -14025.704} C_VEL
LIN {X 0,Y 340.86,Z 159.65,A -85,B 0,C 180,E1 -14029.306,E2 -14029.306} C_VEL
LIN {X 0,Y 341.064,Z 159.605,A -85,B 0,C 180,E1 -14032.898,E2 -14032.898} C_VEL
LIN {X 0,Y 341.16,Z 159.611,A -85,B 0,C 180,E1 -14037.639,E2 -14037.639} C_VEL
LIN {X 0,Y 341.306,Z 159.572,A -85,B 0,C 180,E1 -14040,E2 -14040} C_VEL
LIN {X 0,Y 341.16,Z 159.607,A -85,B 0,C 180,E1 -14042.361,E2 -14042.361} C_VEL
LIN {X 0,Y 341.064,Z 159.602,A -85,B 0,C 180,E1 -14047.102,E2 -14047.102} C_VEL
LIN {X 0,Y 340.86,Z 159.644,A -85,B 0,C 180,E1 -14050.694,E2 -14050.694} C_VEL
LIN {X 0,Y 340.852,Z 159.635,A -85,B 0,C 180,E1 -14054.325,E2 -14054.325} C_VEL
LIN {X 0,Y 340.826,Z 159.635,A -85,B 0,C 180,E1 -14058.467,E2 -14058.467} C_VEL
LIN {X 0,Y 340.743,Z 159.663,A -85,B 0,C 180,E1 -14061.857,E2 -14061.857} C_VEL
LIN {X 0,Y 340.762,Z 159.653,A -85,B 0,C 180,E1 -14065.665,E2 -14065.665} C_VEL
LIN {X 0,Y 340.718,Z 159.662,A -85,B 0,C 180,E1 -14068.322,E2 -14068.322} C_VEL
LIN {X 0,Y 340.688,Z 159.67,A -85,B 0,C 180,E1 -14071.046,E2 -14071.046} C_VEL
LIN {X 0,Y 340.709,Z 159.665,A -85,B 0,C 180,E1 -14075.28,E2 -14075.28} C_VEL
LIN {X 0,Y 340.703,Z 159.65,A -85,B 0,C 180,E1 -14078.388,E2 -14078.388} C_VEL
LIN {X 0,Y 340.691,Z 159.646,A -85,B 0,C 180,E1 -14082.047,E2 -14082.047} C_VEL
LIN {X 0,Y 340.714,Z 159.671,A -85,B 0,C 180,E1 -14085.469,E2 -14085.469} C_VEL
LIN {X 0,Y 340.754,Z 159.807,A -85,B 0,C 180,E1 -14088.205,E2 -14088.205} C_VEL
LIN {X 0,Y 345.802,Z 177.082,A -85,B 0,C 180,E1 -14091.486,E2 -14091.486} C_VEL
LIN {X 0,Y 351.154,Z 195.319,A -85,B 0,C 180,E1 -14094.751,E2 -14094.751} C_VEL
LIN {X 0,Y 353.403,Z 203.668,A -85,B 0,C 180,E1 -14096.166,E2 -14096.166} C_VEL
LIN {X 0,Y 353.021,Z 206.577,A -85,B 0,C 180,E1 -14096.553,E2 -14096.553} C_VEL
LIN {X 0,Y 353.878,Z 218.433,A -85,B 0,C 180,E1 -14097.19,E2 -14097.19} C_VEL
LIN {X 0,Y 359.896,Z 271.118,A -85,B 0,C 180,E1 -14098.995,E2 -14098.995} C_VEL
LIN {X 0,Y 360.244,Z 275.932,A -85,B 0,C 180,E1 -14099.137,E2 -14099.137} C_VEL
LIN {X 0,Y 356.961,Z 392.464,A -85,B 0,C 180,E1 -14101.483,E2 -14101.483} C_VEL
LIN {X 0,Y 355.98,Z 407.424,A -85,B 0,C 180,E1 -14101.96,E2 -14101.96} C_VEL
LIN {X 0,Y 354.586,Z 422.118,A -85,B 0,C 180,E1 -14102.642,E2 -14102.642} C_VEL
LIN {X 0,Y 352.807,Z 436.675,A -85,B 0,C 180,E1 -14103.549,E2 -14103.549} C_VEL
LIN {X 0,Y 351.122,Z 449.542,A -85,B 0,C 180,E1 -14104.583,E2 -14104.583} C_VEL
LIN {X 0,Y 348.88,Z 463.203,A -85,B 0,C 180,E1 -14105.927,E2 -14105.927} C_VEL
LIN {X 0,Y 346.78,Z 476.132,A -85,B 0,C 180,E1 -14107.511,E2 -14107.511} C_VEL
LIN {X 0,Y 344.963,Z 486.96,A -85,B 0,C 180,E1 -14109.114,E2 -14109.114} C_VEL
LIN {X 0,Y 343.381,Z 496.998,A -85,B 0,C 180,E1 -14110.886,E2 -14110.886} C_VEL
LIN {X 0,Y 341.769,Z 506.816,A -85,B 0,C 180,E1 -14112.962,E2 -14112.962} C_VEL
LIN {X 0,Y 340.711,Z 515.023,A -85,B 0,C 180,E1 -14115.06,E2 -14115.06} C_VEL
LIN {X 0,Y 339.99,Z 520.915,A -85,B 0,C 180,E1 -14116.859,E2 -14116.859} C_VEL
LIN {X 0,Y 339.479,Z 527.393,A -85,B 0,C 180,E1 -14119.263,E2 -14119.263} C_VEL
LIN {X 0,Y 339.373,Z 532.42,A -85,B 0,C 180,E1 -14121.667,E2 -14121.667} C_VEL
LIN {X 0,Y 339.473,Z 536.113,A -85,B 0,C 180,E1 -14124.06,E2 -14124.06} C_VEL
LIN {X 0,Y 339.57,Z 538.545,A -85,B 0,C 180,E1 -14126.442,E2 -14126.442} C_VEL
LIN {X 0,Y 339.754,Z 539.778,A -85,B 0,C 180,E1 -14128.816,E2 -14128.816} C_VEL
LIN {X 0,Y 339.748,Z 539.776,A -85,B 0,C 180,E1 -14131.187,E2 -14131.187} C_VEL
LIN {X 0,Y 339.57,Z 538.538,A -85,B 0,C 180,E1 -14133.561,E2 -14133.561} C_VEL
LIN {X 0,Y 339.494,Z 536.099,A -85,B 0,C 180,E1 -14135.943,E2 -14135.943} C_VEL
LIN {X 0,Y 339.392,Z 532.391,A -85,B 0,C 180,E1 -14138.336,E2 -14138.336} C_VEL
LIN {X 0,Y 339.514,Z 527.352,A -85,B 0,C 180,E1 -14140.738,E2 -14140.738} C_VEL
LIN {X 0,Y 340.034,Z 520.87,A -85,B 0,C 180,E1 -14143.143,E2 -14143.143} C_VEL
LIN {X 0,Y 340.995,Z 512.754,A -85,B 0,C 180,E1 -14145.543,E2 -14145.543} C_VEL
LIN {X 0,Y 342.265,Z 504.117,A -85,B 0,C 180,E1 -14147.632,E2 -14147.632} C_VEL
LIN {X 0,Y 343.815,Z 494.511,A -85,B 0,C 180,E1 -14149.567,E2 -14149.567} C_VEL
LIN {X 0,Y 345.271,Z 485.046,A -85,B 0,C 180,E1 -14151.182,E2 -14151.182} C_VEL
LIN {X 0,Y 347.156,Z 473.836,A -85,B 0,C 180,E1 -14152.78,E2 -14152.78} C_VEL
LIN {X 0,Y 349.123,Z 461.737,A -85,B 0,C 180,E1 -14154.216,E2 -14154.216} C_VEL
LIN {X 0,Y 351.11,Z 449.04,A -85,B 0,C 180,E1 -14155.451,E2 -14155.451} C_VEL
LIN {X 0,Y 352.998,Z 435.333,A -85,B 0,C 180,E1 -14156.526,E2 -14156.526} C_VEL
LIN {X 0,Y 354.791,Z 421.501,A -85,B 0,C 180,E1 -14157.424,E2 -14157.424} C_VEL
LIN {X 0,Y 356.965,Z 407.657,A -85,B 0,C 180,E1 -14158.279,E2 -14158.279} C_VEL
LIN {X 0,Y 358.949,Z 391.912,A -85,B 0,C 180,E1 -14159.027,E2 -14159.027} C_VEL
LIN {X 0,Y 360.499,Z 374.784,A -85,B 0,C 180,E1 -14159.61,E2 -14159.61} C_VEL
LIN {X 0,Y 365.234,Z 315.472,A -85,B 0,C 180,E1 -14161.431,E2 -14161.431} C_VEL
LIN {X 0,Y 368.82,Z 275.74,A -85,B 0,C 180,E1 -14162.734,E2 -14162.734} C_VEL
LIN {X 0,Y 368.484,Z 259.938,A -85,B 0,C 180,E1 -14163.604,E2 -14163.604} C_VEL
LIN {X 0,Y 367.446,Z 245.207,A -85,B 0,C 180,E1 -14164.64,E2 -14164.64} C_VEL
LIN {X 0,Y 365.832,Z 228.919,A -85,B 0,C 180,E1 -14166.023,E2 -14166.023} C_VEL
LIN {X 0,Y 367.198,Z 225.136,A -85,B 0,C 180,E1 -14166.699,E2 -14166.699} C_VEL
LIN {X 0,Y 366.888,Z 222.282,A -85,B 0,C 180,E1 -14167.563,E2 -14167.563} C_VEL
LIN {X 0,Y 365.538,Z 216.619,A -85,B 0,C 180,E1 -14169.731,E2 -14169.731} C_VEL
LIN {X 0,Y 364.685,Z 213.4,A -85,B 0,C 180,E1 -14171.272,E2 -14171.272} C_VEL
LIN {X 0,Y 363.855,Z 210.958,A -85,B 0,C 180,E1 -14172.779,E2 -14172.779} C_VEL
LIN {X 0,Y 363.135,Z 209.134,A -85,B 0,C 180,E1 -14174.268,E2 -14174.268} C_VEL
LIN {X 0,Y 362.532,Z 207.797,A -85,B 0,C 180,E1 -14175.832,E2 -14175.832} C_VEL
LIN {X 0,Y 362.065,Z 206.972,A -85,B 0,C 180,E1 -14177.53,E2 -14177.53} C_VEL
LIN {X 0,Y 361.659,Z 206.976,A -85,B 0,C 180,E1 -14180.113,E2 -14180.113} C_VEL
LIN {X 0,Y 361.609,Z 207.588,A -85,B 0,C 180,E1 -14181.543,E2 -14181.543} C_VEL
LIN {X 0,Y 361.648,Z 208.62,A -85,B 0,C 180,E1 -14182.956,E2 -14182.956} C_VEL
LIN {X 0,Y 361.988,Z 211.781,A -85,B 0,C 180,E1 -14185.734,E2 -14185.734} C_VEL
LIN {X 0,Y 362.398,Z 216.13,A -85,B 0,C 180,E1 -14188.281,E2 -14188.281} C_VEL
LIN {X 0,Y 364.115,Z 219.581,A -85,B 0,C 180,E1 -14189.165,E2 -14189.165} C_VEL
LIN {X 0,Y 366.143,Z 223.25,A -85,B 0,C 180,E1 -14190.007,E2 -14190.007} C_VEL
LIN {X 0,Y 367.9,Z 226.945,A -85,B 0,C 180,E1 -14190.719,E2 -14190.719} C_VEL
LIN {X 0,Y 370.19,Z 238.446,A -85,B 0,C 180,E1 -14192.035,E2 -14192.035} C_VEL
LIN {X 0,Y 371.154,Z 245.017,A -85,B 0,C 180,E1 -14192.662,E2 -14192.662} C_VEL
LIN {X 0,Y 361.448,Z 327.376,A -85,B 0,C 180,E1 -14195.901,E2 -14195.901} C_VEL
LIN {X 0,Y 360.153,Z 343.363,A -85,B 0,C 180,E1 -14196.657,E2 -14196.657} C_VEL
LIN {X 0,Y 358.756,Z 356.905,A -85,B 0,C 180,E1 -14197.515,E2 -14197.515} C_VEL
LIN {X 0,Y 356.949,Z 370.817,A -85,B 0,C 180,E1 -14198.639,E2 -14198.639} C_VEL
LIN {X 0,Y 355.111,Z 382.999,A -85,B 0,C 180,E1 -14199.887,E2 -14199.887} C_VEL
LIN {X 0,Y 353.266,Z 394.097,A -85,B 0,C 180,E1 -14201.289,E2 -14201.289} C_VEL
LIN {X 0,Y 351.37,Z 404.116,A -85,B 0,C 180,E1 -14202.841,E2 -14202.841} C_VEL
LIN {X 0,Y 349.547,Z 413.043,A -85,B 0,C 180,E1 -14204.55,E2 -14204.55} C_VEL
LIN {X 0,Y 347.724,Z 420.806,A -85,B 0,C 180,E1 -14206.374,E2 -14206.374} C_VEL
LIN {X 0,Y 346.105,Z 427.143,A -85,B 0,C 180,E1 -14208.284,E2 -14208.284} C_VEL
LIN {X 0,Y 344.859,Z 431.617,A -85,B 0,C 180,E1 -14210.025,E2 -14210.025} C_VEL
LIN {X 0,Y 343.719,Z 435.031,A -85,B 0,C 180,E1 -14211.771,E2 -14211.771} C_VEL
LIN {X 0,Y 343.12,Z 436.69,A -85,B 0,C 180,E1 -14212.941,E2 -14212.941} C_VEL
LIN {X 0,Y 342.647,Z 437.924,A -85,B 0,C 180,E1 -14214.114,E2 -14214.114} C_VEL
LIN {X 0,Y 342.285,Z 438.739,A -85,B 0,C 180,E1 -14215.289,E2 -14215.289} C_VEL
LIN {X 0,Y 341.881,Z 439.129,A -85,B 0,C 180,E1 -14216.464,E2 -14216.464} C_VEL
LIN {X 0,Y 341.614,Z 439.071,A -85,B 0,C 180,E1 -14217.642,E2 -14217.642} C_VEL
LIN {X 0,Y 341.274,Z 438.624,A -85,B 0,C 180,E1 -14218.82,E2 -14218.82} C_VEL
LIN {X 0,Y 340.999,Z 437.764,A -85,B 0,C 180,E1 -14220,E2 -14220} C_VEL
LIN {X 0,Y 341.014,Z 436.439,A -85,B 0,C 180,E1 -14221.181,E2 -14221.181} C_VEL
LIN {X 0,Y 340.912,Z 433.66,A -85,B 0,C 180,E1 -14222.954,E2 -14222.954} C_VEL
LIN {X 0,Y 340.818,Z 429.853,A -85,B 0,C 180,E1 -14224.731,E2 -14224.731} C_VEL
LIN {X 0,Y 341.166,Z 424.911,A -85,B 0,C 180,E1 -14226.506,E2 -14226.506} C_VEL
LIN {X 0,Y 341.452,Z 418.738,A -85,B 0,C 180,E1 -14228.284,E2 -14228.284} C_VEL
LIN {X 0,Y 341.835,Z 411.119,A -85,B 0,C 180,E1 -14230.065,E2 -14230.065} C_VEL
LIN {X 0,Y 342.467,Z 401.811,A -85,B 0,C 180,E1 -14231.842,E2 -14231.842} C_VEL
LIN {X 0,Y 343.097,Z 391.352,A -85,B 0,C 180,E1 -14233.474,E2 -14233.474} C_VEL
LIN {X 0,Y 343.819,Z 379.723,A -85,B 0,C 180,E1 -14234.956,E2 -14234.956} C_VEL
LIN {X 0,Y 344.568,Z 367.155,A -85,B 0,C 180,E1 -14236.252,E2 -14236.252} C_VEL
LIN {X 0,Y 345.184,Z 353.088,A -85,B 0,C 180,E1 -14237.4,E2 -14237.4} C_VEL
LIN {X 0,Y 345.737,Z 340.1,A -85,B 0,C 180,E1 -14238.212,E2 -14238.212} C_VEL
LIN {X 0,Y 346.121,Z 327.462,A -85,B 0,C 180,E1 -14238.805,E2 -14238.805} C_VEL
LIN {X 0,Y 346.737,Z 302.72,A -85,B 0,C 180,E1 -14239.577,E2 -14239.577} C_VEL
LIN {X 0,Y 349.272,Z 228.029,A -85,B 0,C 180,E1 -14241.748,E2 -14241.748} C_VEL
LIN {X 0,Y 345.551,Z 203.586,A -85,B 0,C 180,E1 -14242.691,E2 -14242.691} C_VEL
LIN {X 0,Y 346.95,Z 188.586,A -85,B 0,C 180,E1 -14245.818,E2 -14245.818} C_VEL
LIN {X 0,Y 345.934,Z 182.462,A -85,B 0,C 180,E1 -14247.23,E2 -14247.23} C_VEL
LIN {X 0,Y 343.06,Z 169.574,A -85,B 0,C 180,E1 -14250.313,E2 -14250.313} C_VEL
LIN {X 0,Y 340.731,Z 159.668,A -85,B 0,C 180,E1 -14252.782,E2 -14252.782} C_VEL
LIN {X 0,Y 340.714,Z 159.669,A -85,B 0,C 180,E1 -14256.44,E2 -14256.44} C_VEL
LIN {X 0,Y 340.684,Z 159.66,A -85,B 0,C 180,E1 -14259.755,E2 -14259.755} C_VEL
LIN {X 0,Y 340.68,Z 159.668,A -85,B 0,C 180,E1 -14262.904,E2 -14262.904} C_VEL
LIN {X 0,Y 340.674,Z 159.672,A -85,B 0,C 180,E1 -14266.223,E2 -14266.223} C_VEL
LIN {X 0,Y 340.693,Z 159.667,A -85,B 0,C 180,E1 -14269.752,E2 -14269.752} C_VEL
LIN {X 0,Y 340.71,Z 159.671,A -85,B 0,C 180,E1 -14273.258,E2 -14273.258} C_VEL
LIN {X 0,Y 340.744,Z 159.831,A -85,B 0,C 180,E1 -14273.552,E2 -14273.552} C_VEL
LIN {X 0,Y 345.528,Z 172.961,A -85,B 0,C 180,E1 -14276.18,E2 -14276.18} C_VEL
LIN {X 0,Y 354.875,Z 190.644,A -85,B 0,C 180,E1 -14277.633,E2 -14277.633} C_VEL
LIN {X 0,Y 362.325,Z 206.514,A -85,B 0,C 180,E1 -14278.754,E2 -14278.754} C_VEL
LIN {X 0,Y 362.519,Z 209.427,A -85,B 0,C 180,E1 -14278.84,E2 -14278.84} C_VEL
LIN {X 0,Y 358.757,Z 339.711,A -85,B 0,C 180,E1 -14281.476,E2 -14281.476} C_VEL
LIN {X 0,Y 358.127,Z 354.246,A -85,B 0,C 180,E1 -14281.971,E2 -14281.971} C_VEL
LIN {X 0,Y 357.195,Z 367.898,A -85,B 0,C 180,E1 -14282.628,E2 -14282.628} C_VEL
LIN {X 0,Y 356.051,Z 381.247,A -85,B 0,C 180,E1 -14283.474,E2 -14283.474} C_VEL
LIN {X 0,Y 354.427,Z 395.371,A -85,B 0,C 180,E1 -14284.607,E2 -14284.607} C_VEL
LIN {X 0,Y 352.647,Z 408.213,A -85,B 0,C 180,E1 -14285.885,E2 -14285.885} C_VEL
LIN {X 0,Y 350.692,Z 420.414,A -85,B 0,C 180,E1 -14287.362,E2 -14287.362} C_VEL
LIN {X 0,Y 348.926,Z 431.825,A -85,B 0,C 180,E1 -14289.051,E2 -14289.051} C_VEL
LIN {X 0,Y 347.067,Z 441.719,A -85,B 0,C 180,E1 -14290.787,E2 -14290.787} C_VEL
LIN {X 0,Y 345.172,Z 451.615,A -85,B 0,C 180,E1 -14292.888,E2 -14292.888} C_VEL
LIN {X 0,Y 343.58,Z 460.373,A -85,B 0,C 180,E1 -14295.184,E2 -14295.184} C_VEL
LIN {X 0,Y 342.212,Z 467.628,A -85,B 0,C 180,E1 -14297.546,E2 -14297.546} C_VEL
LIN {X 0,Y 341.212,Z 473.371,A -85,B 0,C 180,E1 -14299.916,E2 -14299.916} C_VEL
LIN {X 0,Y 340.542,Z 477.53,A -85,B 0,C 180,E1 -14302.143,E2 -14302.143} C_VEL
LIN {X 0,Y 340.084,Z 480.208,A -85,B 0,C 180,E1 -14304.068,E2 -14304.068} C_VEL
LIN {X 0,Y 340.066,Z 481.474,A -85,B 0,C 180,E1 -14305.257,E2 -14305.257} C_VEL
LIN {X 0,Y 339.721,Z 483.192,A -85,B 0,C 180,E1 -14307.627,E2 -14307.627} C_VEL
LIN {X 0,Y 339.609,Z 483.786,A -85,B 0,C 180,E1 -14309.998,E2 -14309.998} C_VEL
LIN {X 0,Y 339.719,Z 483.231,A -85,B 0,C 180,E1 -14312.37,E2 -14312.37} C_VEL
LIN {X 0,Y 340.059,Z 481.568,A -85,B 0,C 180,E1 -14314.74,E2 -14314.74} C_VEL
LIN {X 0,Y 340.406,Z 478.398,A -85,B 0,C 180,E1 -14317.381,E2 -14317.381} C_VEL
LIN {X 0,Y 340.99,Z 474.788,A -85,B 0,C 180,E1 -14319.489,E2 -14319.489} C_VEL
LIN {X 0,Y 341.872,Z 469.468,A -85,B 0,C 180,E1 -14321.861,E2 -14321.861} C_VEL
LIN {X 0,Y 342.045,Z 468.505,A -85,B 0,C 180,E1 -14322.228,E2 -14322.228} C_VEL
LIN {X 0,Y 341.839,Z 466.154,A -85,B 0,C 180,E1 -14323.137,E2 -14323.137} C_VEL
LIN {X 0,Y 339.799,Z 462.194,A -85,B 0,C 180,E1 -14324.632,E2 -14324.632} C_VEL
LIN {X 0,Y 337.9,Z 457.774,A -85,B 0,C 180,E1 -14326.102,E2 -14326.102} C_VEL
LIN {X 0,Y 337.906,Z 454.662,A -85,B 0,C 180,E1 -14326.956,E2 -14326.956} C_VEL
LIN {X 0,Y 339.764,Z 445.713,A -85,B 0,C 180,E1 -14329.012,E2 -14329.012} C_VEL
LIN {X 0,Y 341.56,Z 436.479,A -85,B 0,C 180,E1 -14330.788,E2 -14330.788} C_VEL
LIN {X 0,Y 343.456,Z 425.51,A -85,B 0,C 180,E1 -14332.56,E2 -14332.56} C_VEL
LIN {X 0,Y 345.514,Z 413.431,A -85,B 0,C 180,E1 -14334.163,E2 -14334.163} C_VEL
LIN {X 0,Y 347.561,Z 400.069,A -85,B 0,C 180,E1 -14335.607,E2 -14335.607} C_VEL
LIN {X 0,Y 349.228,Z 386.972,A -85,B 0,C 180,E1 -14336.76,E2 -14336.76} C_VEL
LIN {X 0,Y 350.719,Z 372.204,A -85,B 0,C 180,E1 -14337.787,E2 -14337.787} C_VEL
LIN {X 0,Y 351.709,Z 358.829,A -85,B 0,C 180,E1 -14338.507,E2 -14338.507} C_VEL
LIN {X 0,Y 352.514,Z 343.969,A -85,B 0,C 180,E1 -14339.073,E2 -14339.073} C_VEL
LIN {X 0,Y 353.2,Z 321.667,A -85,B 0,C 180,E1 -14339.583,E2 -14339.583} C_VEL
LIN {X 0,Y 356.468,Z 209.006,A -85,B 0,C 180,E1 -14341.883,E2 -14341.883} C_VEL
LIN {X 0,Y 347.415,Z 190.041,A -85,B 0,C 180,E1 -14343.295,E2 -14343.295} C_VEL
LIN {X 0,Y 338.494,Z 173.507,A -85,B 0,C 180,E1 -14344.75,E2 -14344.75} C_VEL
LIN {X 0,Y 333.653,Z 160.549,A -85,B 0,C 180,E1 -14347.447,E2 -14347.447} C_VEL
LIN {X 0,Y 333.641,Z 160.524,A -85,B 0,C 180,E1 -14350.766,E2 -14350.766} C_VEL
LIN {X 0,Y 333.602,Z 160.547,A -85,B 0,C 180,E1 -14354.252,E2 -14354.252} C_VEL
LIN {X 0,Y 333.666,Z 160.539,A -85,B 0,C 180,E1 -14357.622,E2 -14357.622} C_VEL
LIN {X 0,Y 333.669,Z 160.537,A -85,B 0,C 180,E1 -14361.195,E2 -14361.195} C_VEL
LIN {X 0,Y 333.677,Z 160.534,A -85,B 0,C 180,E1 -14365.225,E2 -14365.225} C_VEL
LIN {X 0,Y 333.636,Z 160.55,A -85,B 0,C 180,E1 -14368.222,E2 -14368.222} C_VEL
LIN {X 0,Y 333.703,Z 160.53,A -85,B 0,C 180,E1 -14371.027,E2 -14371.027} C_VEL
LIN {X 0,Y 333.726,Z 160.534,A -85,B 0,C 180,E1 -14373.753,E2 -14373.753} C_VEL
LIN {X 0,Y 333.709,Z 160.541,A -85,B 0,C 180,E1 -14377.913,E2 -14377.913} C_VEL
LIN {X 0,Y 333.783,Z 160.516,A -85,B 0,C 180,E1 -14381.589,E2 -14381.589} C_VEL
LIN {X 0,Y 333.798,Z 160.521,A -85,B 0,C 180,E1 -14385.576,E2 -14385.576} C_VEL
LIN {X 0,Y 333.823,Z 160.523,A -85,B 0,C 180,E1 -14389.078,E2 -14389.078} C_VEL
LIN {X 0,Y 334.014,Z 160.484,A -85,B 0,C 180,E1 -14392.747,E2 -14392.747} C_VEL
LIN {X 0,Y 333.802,Z 160.52,A -85,B 0,C 180,E1 -14395.169,E2 -14395.169} C_VEL
LIN {X 0,Y 334.097,Z 160.491,A -85,B 0,C 180,E1 -14397.589,E2 -14397.589} C_VEL
LIN {X 0,Y 334.257,Z 160.45,A -85,B 0,C 180,E1 -14400,E2 -14400} C_VEL
LIN {X 0,Y 334.097,Z 160.487,A -85,B 0,C 180,E1 -14402.411,E2 -14402.411} C_VEL
LIN {X 0,Y 334.014,Z 160.481,A -85,B 0,C 180,E1 -14407.253,E2 -14407.253} C_VEL
LIN {X 0,Y 333.823,Z 160.519,A -85,B 0,C 180,E1 -14410.922,E2 -14410.922} C_VEL
LIN {X 0,Y 333.797,Z 160.517,A -85,B 0,C 180,E1 -14414.635,E2 -14414.635} C_VEL
LIN {X 0,Y 333.785,Z 160.511,A -85,B 0,C 180,E1 -14418.655,E2 -14418.655} C_VEL
LIN {X 0,Y 333.682,Z 160.544,A -85,B 0,C 180,E1 -14422.279,E2 -14422.279} C_VEL
LIN {X 0,Y 333.725,Z 160.534,A -85,B 0,C 180,E1 -14426.247,E2 -14426.247} C_VEL
LIN {X 0,Y 333.68,Z 160.533,A -85,B 0,C 180,E1 -14428.975,E2 -14428.975} C_VEL
LIN {X 0,Y 333.633,Z 160.549,A -85,B 0,C 180,E1 -14432.588,E2 -14432.588} C_VEL
LIN {X 0,Y 333.668,Z 160.548,A -85,B 0,C 180,E1 -14436.14,E2 -14436.14} C_VEL
LIN {X 0,Y 333.638,Z 160.512,A -85,B 0,C 180,E1 -14439.193,E2 -14439.193} C_VEL
LIN {X 0,Y 333.625,Z 160.535,A -85,B 0,C 180,E1 -14442.501,E2 -14442.501} C_VEL
LIN {X 0,Y 333.661,Z 160.548,A -85,B 0,C 180,E1 -14445.968,E2 -14445.968} C_VEL
LIN {X 0,Y 333.722,Z 160.641,A -85,B 0,C 180,E1 -14447.682,E2 -14447.682} C_VEL
LIN {X 0,Y 338.709,Z 177.775,A -85,B 0,C 180,E1 -14451.02,E2 -14451.02} C_VEL
LIN {X 0,Y 344.263,Z 196.788,A -85,B 0,C 180,E1 -14454.491,E2 -14454.491} C_VEL
LIN {X 0,Y 346.224,Z 203.848,A -85,B 0,C 180,E1 -14455.691,E2 -14455.691} C_VEL
LIN {X 0,Y 346.866,Z 206.774,A -85,B 0,C 180,E1 -14455.906,E2 -14455.906} C_VEL
LIN {X 0,Y 347.649,Z 218.079,A -85,B 0,C 180,E1 -14456.529,E2 -14456.529} C_VEL
LIN {X 0,Y 352.702,Z 261.826,A -85,B 0,C 180,E1 -14458.086,E2 -14458.086} C_VEL
LIN {X 0,Y 354.13,Z 276.559,A -85,B 0,C 180,E1 -14458.569,E2 -14458.569} C_VEL
LIN {X 0,Y 350.74,Z 391.982,A -85,B 0,C 180,E1 -14460.93,E2 -14460.93} C_VEL
LIN {X 0,Y 349.739,Z 406.897,A -85,B 0,C 180,E1 -14461.414,E2 -14461.414} C_VEL
LIN {X 0,Y 348.291,Z 421.57,A -85,B 0,C 180,E1 -14462.105,E2 -14462.105} C_VEL
LIN {X 0,Y 346.452,Z 435.908,A -85,B 0,C 180,E1 -14463.008,E2 -14463.008} C_VEL
LIN {X 0,Y 344.587,Z 449.555,A -85,B 0,C 180,E1 -14464.125,E2 -14464.125} C_VEL
LIN {X 0,Y 342.384,Z 462.63,A -85,B 0,C 180,E1 -14465.441,E2 -14465.441} C_VEL
LIN {X 0,Y 340.334,Z 474.473,A -85,B 0,C 180,E1 -14466.901,E2 -14466.901} C_VEL
LIN {X 0,Y 338.244,Z 486.374,A -85,B 0,C 180,E1 -14468.68,E2 -14468.68} C_VEL
LIN {X 0,Y 336.611,Z 496.412,A -85,B 0,C 180,E1 -14470.487,E2 -14470.487} C_VEL
LIN {X 0,Y 334.912,Z 506.228,A -85,B 0,C 180,E1 -14472.602,E2 -14472.602} C_VEL
LIN {X 0,Y 333.727,Z 514.429,A -85,B 0,C 180,E1 -14474.739,E2 -14474.739} C_VEL
LIN {X 0,Y 332.805,Z 522.095,A -85,B 0,C 180,E1 -14477.191,E2 -14477.191} C_VEL
LIN {X 0,Y 332.349,Z 528.204,A -85,B 0,C 180,E1 -14479.647,E2 -14479.647} C_VEL
LIN {X 0,Y 332.299,Z 532.908,A -85,B 0,C 180,E1 -14482.1,E2 -14482.1} C_VEL
LIN {X 0,Y 332.384,Z 535.524,A -85,B 0,C 180,E1 -14483.933,E2 -14483.933} C_VEL
LIN {X 0,Y 332.475,Z 537.958,A -85,B 0,C 180,E1 -14486.366,E2 -14486.366} C_VEL
LIN {X 0,Y 332.673,Z 539.193,A -85,B 0,C 180,E1 -14488.791,E2 -14488.791} C_VEL
LIN {X 0,Y 332.667,Z 539.191,A -85,B 0,C 180,E1 -14491.212,E2 -14491.212} C_VEL
LIN {X 0,Y 332.476,Z 537.951,A -85,B 0,C 180,E1 -14493.637,E2 -14493.637} C_VEL
LIN {X 0,Y 332.439,Z 535.004,A -85,B 0,C 180,E1 -14496.479,E2 -14496.479} C_VEL
LIN {X 0,Y 332.308,Z 530.692,A -85,B 0,C 180,E1 -14499.128,E2 -14499.128} C_VEL
LIN {X 0,Y 332.598,Z 525.295,A -85,B 0,C 180,E1 -14501.582,E2 -14501.582} C_VEL
LIN {X 0,Y 333.304,Z 517.875,A -85,B 0,C 180,E1 -14504.218,E2 -14504.218} C_VEL
LIN {X 0,Y 334.365,Z 509.878,A -85,B 0,C 180,E1 -14506.486,E2 -14506.486} C_VEL
LIN {X 0,Y 335.86,Z 500.773,A -85,B 0,C 180,E1 -14508.611,E2 -14508.611} C_VEL
LIN {X 0,Y 337.465,Z 490.937,A -85,B 0,C 180,E1 -14510.524,E2 -14510.524} C_VEL
LIN {X 0,Y 339.238,Z 480.558,A -85,B 0,C 180,E1 -14512.217,E2 -14512.217} C_VEL
LIN {X 0,Y 341.343,Z 468.644,A -85,B 0,C 180,E1 -14513.834,E2 -14513.834} C_VEL
LIN {X 0,Y 343.321,Z 457.066,A -85,B 0,C 180,E1 -14515.137,E2 -14515.137} C_VEL
LIN {X 0,Y 345.339,Z 443.754,A -85,B 0,C 180,E1 -14516.37,E2 -14516.37} C_VEL
LIN {X 0,Y 347.971,Z 426.816,A -85,B 0,C 180,E1 -14517.681,E2 -14517.681} C_VEL
LIN {X 0,Y 350.675,Z 411.436,A -85,B 0,C 180,E1 -14518.752,E2 -14518.752} C_VEL
LIN {X 0,Y 353.025,Z 395.278,A -85,B 0,C 180,E1 -14519.603,E2 -14519.603} C_VEL
LIN {X 0,Y 354.823,Z 378.233,A -85,B 0,C 180,E1 -14520.256,E2 -14520.256} C_VEL
LIN {X 0,Y 360.347,Z 315.173,A -85,B 0,C 180,E1 -14522.255,E2 -14522.255} C_VEL
LIN {X 0,Y 364.113,Z 276.619,A -85,B 0,C 180,E1 -14523.557,E2 -14523.557} C_VEL
LIN {X 0,Y 363.965,Z 260.836,A -85,B 0,C 180,E1 -14524.474,E2 -14524.474} C_VEL
LIN {X 0,Y 363.161,Z 247.17,A -85,B 0,C 180,E1 -14525.492,E2 -14525.492} C_VEL
LIN {X 0,Y 361.922,Z 232.318,A -85,B 0,C 180,E1 -14526.789,E2 -14526.789} C_VEL
LIN {X 0,Y 361.606,Z 228.14,A -85,B 0,C 180,E1 -14527.233,E2 -14527.233} C_VEL
LIN {X 0,Y 360.511,Z 222.709,A -85,B 0,C 180,E1 -14529.2,E2 -14529.2} C_VEL
LIN {X 0,Y 359.492,Z 218.406,A -85,B 0,C 180,E1 -14531.179,E2 -14531.179} C_VEL
LIN {X 0,Y 358.265,Z 214.926,A -85,B 0,C 180,E1 -14533.463,E2 -14533.463} C_VEL
LIN {X 0,Y 357.578,Z 213.267,A -85,B 0,C 180,E1 -14535.038,E2 -14535.038} C_VEL
LIN {X 0,Y 357.009,Z 212.11,A -85,B 0,C 180,E1 -14536.752,E2 -14536.752} C_VEL
LIN {X 0,Y 356.641,Z 211.612,A -85,B 0,C 180,E1 -14538.491,E2 -14538.491} C_VEL
LIN {X 0,Y 356.332,Z 212.024,A -85,B 0,C 180,E1 -14540.866,E2 -14540.866} C_VEL
LIN {X 0,Y 356.291,Z 212.844,A -85,B 0,C 180,E1 -14542.303,E2 -14542.303} C_VEL
LIN {X 0,Y 356.463,Z 215.655,A -85,B 0,C 180,E1 -14545.127,E2 -14545.127} C_VEL
LIN {X 0,Y 356.769,Z 217.831,A -85,B 0,C 180,E1 -14546.582,E2 -14546.582} C_VEL
LIN {X 0,Y 359.956,Z 223.419,A -85,B 0,C 180,E1 -14548.251,E2 -14548.251} C_VEL
LIN {X 0,Y 362.441,Z 228.099,A -85,B 0,C 180,E1 -14549.396,E2 -14549.396} C_VEL
LIN {X 0,Y 364.126,Z 231.743,A -85,B 0,C 180,E1 -14550.144,E2 -14550.144} C_VEL
LIN {X 0,Y 366.252,Z 244.018,A -85,B 0,C 180,E1 -14551.564,E2 -14551.564} C_VEL
LIN {X 0,Y 366.595,Z 246.859,A -85,B 0,C 180,E1 -14551.84,E2 -14551.84} C_VEL
LIN {X 0,Y 356.493,Z 327.07,A -85,B 0,C 180,E1 -14555.077,E2 -14555.077} C_VEL
LIN {X 0,Y 354.934,Z 344.19,A -85,B 0,C 180,E1 -14555.9,E2 -14555.9} C_VEL
LIN {X 0,Y 353.349,Z 358.149,A -85,B 0,C 180,E1 -14556.801,E2 -14556.801} C_VEL
LIN {X 0,Y 351.362,Z 372.291,A -85,B 0,C 180,E1 -14557.973,E2 -14557.973} C_VEL
LIN {X 0,Y 349.181,Z 385.52,A -85,B 0,C 180,E1 -14559.377,E2 -14559.377} C_VEL
LIN {X 0,Y 347.234,Z 396.31,A -85,B 0,C 180,E1 -14560.798,E2 -14560.798} C_VEL
LIN {X 0,Y 345.364,Z 405.278,A -85,B 0,C 180,E1 -14562.227,E2 -14562.227} C_VEL
LIN {X 0,Y 343.393,Z 414.167,A -85,B 0,C 180,E1 -14563.962,E2 -14563.962} C_VEL
LIN {X 0,Y 341.504,Z 421.498,A -85,B 0,C 180,E1 -14565.703,E2 -14565.703} C_VEL
LIN {X 0,Y 339.968,Z 427.381,A -85,B 0,C 180,E1 -14567.464,E2 -14567.464} C_VEL
LIN {X 0,Y 338.438,Z 432.09,A -85,B 0,C 180,E1 -14569.229,E2 -14569.229} C_VEL
LIN {X 0,Y 337.312,Z 435.642,A -85,B 0,C 180,E1 -14571.01,E2 -14571.01} C_VEL
LIN {X 0,Y 336.242,Z 438.183,A -85,B 0,C 180,E1 -14572.796,E2 -14572.796} C_VEL
LIN {X 0,Y 335.747,Z 439.334,A -85,B 0,C 180,E1 -14573.992,E2 -14573.992} C_VEL
LIN {X 0,Y 335.344,Z 440.037,A -85,B 0,C 180,E1 -14575.191,E2 -14575.191} C_VEL
LIN {X 0,Y 334.901,Z 440.321,A -85,B 0,C 180,E1 -14576.391,E2 -14576.391} C_VEL
LIN {X 0,Y 334.617,Z 440.186,A -85,B 0,C 180,E1 -14577.593,E2 -14577.593} C_VEL
LIN {X 0,Y 334.261,Z 439.659,A -85,B 0,C 180,E1 -14578.795,E2 -14578.795} C_VEL
LIN {X 0,Y 333.972,Z 438.706,A -85,B 0,C 180,E1 -14580,E2 -14580} C_VEL
LIN {X 0,Y 333.986,Z 437.266,A -85,B 0,C 180,E1 -14581.206,E2 -14581.206} C_VEL
LIN {X 0,Y 333.872,Z 434.346,A -85,B 0,C 180,E1 -14583.017,E2 -14583.017} C_VEL
LIN {X 0,Y 333.775,Z 430.394,A -85,B 0,C 180,E1 -14584.832,E2 -14584.832} C_VEL
LIN {X 0,Y 334.131,Z 425.293,A -85,B 0,C 180,E1 -14586.643,E2 -14586.643} C_VEL
LIN {X 0,Y 334.495,Z 417.818,A -85,B 0,C 180,E1 -14588.745,E2 -14588.745} C_VEL
LIN {X 0,Y 334.953,Z 409.705,A -85,B 0,C 180,E1 -14590.579,E2 -14590.579} C_VEL
LIN {X 0,Y 335.577,Z 399.789,A -85,B 0,C 180,E1 -14592.396,E2 -14592.396} C_VEL
LIN {X 0,Y 336.254,Z 388.687,A -85,B 0,C 180,E1 -14594.062,E2 -14594.062} C_VEL
LIN {X 0,Y 337.082,Z 376.16,A -85,B 0,C 180,E1 -14595.571,E2 -14595.571} C_VEL
LIN {X 0,Y 337.741,Z 363.388,A -85,B 0,C 180,E1 -14596.819,E2 -14596.819} C_VEL
LIN {X 0,Y 338.482,Z 348.969,A -85,B 0,C 180,E1 -14597.912,E2 -14597.912} C_VEL
LIN {X 0,Y 338.876,Z 335.139,A -85,B 0,C 180,E1 -14598.712,E2 -14598.712} C_VEL
LIN {X 0,Y 339.385,Z 320.18,A -85,B 0,C 180,E1 -14599.31,E2 -14599.31} C_VEL
LIN {X 0,Y 342.399,Z 228.831,A -85,B 0,C 180,E1 -14602.05,E2 -14602.05} C_VEL
LIN {X 0,Y 338.705,Z 203.734,A -85,B 0,C 180,E1 -14603.063,E2 -14603.063} C_VEL
LIN {X 0,Y 340.056,Z 189.643,A -85,B 0,C 180,E1 -14606.052,E2 -14606.052} C_VEL
LIN {X 0,Y 338.329,Z 180.533,A -85,B 0,C 180,E1 -14608.202,E2 -14608.202} C_VEL
LIN {X 0,Y 334.82,Z 165.345,A -85,B 0,C 180,E1 -14611.941,E2 -14611.941} C_VEL
LIN {X 0,Y 333.678,Z 160.548,A -85,B 0,C 180,E1 -14613.204,E2 -14613.204} C_VEL
LIN {X 0,Y 333.669,Z 160.549,A -85,B 0,C 180,E1 -14616.831,E2 -14616.831} C_VEL
LIN {X 0,Y 333.648,Z 160.541,A -85,B 0,C 180,E1 -14620.767,E2 -14620.767} C_VEL
LIN {X 0,Y 333.629,Z 160.543,A -85,B 0,C 180,E1 -14624.255,E2 -14624.255} C_VEL
LIN {X 0,Y 333.648,Z 160.544,A -85,B 0,C 180,E1 -14627.618,E2 -14627.618} C_VEL
LIN {X 0,Y 333.658,Z 160.552,A -85,B 0,C 180,E1 -14631.201,E2 -14631.201} C_VEL
LIN {X 0,Y 333.669,Z 160.609,A -85,B 0,C 180,E1 -14632.721,E2 -14632.721} C_VEL
LIN {X 0,Y 338.563,Z 173.739,A -85,B 0,C 180,E1 -14635.402,E2 -14635.402} C_VEL
LIN {X 0,Y 348.04,Z 191.285,A -85,B 0,C 180,E1 -14636.918,E2 -14636.918} C_VEL
LIN {X 0,Y 355.474,Z 206.917,A -85,B 0,C 180,E1 -14638.078,E2 -14638.078} C_VEL
LIN {X 0,Y 356.485,Z 209.468,A -85,B 0,C 180,E1 -14638.241,E2 -14638.241} C_VEL
LIN {X 0,Y 352.55,Z 340.233,A -85,B 0,C 180,E1 -14640.927,E2 -14640.927} C_VEL
LIN {X 0,Y 351.833,Z 355.675,A -85,B 0,C 180,E1 -14641.465,E2 -14641.465} C_VEL
LIN {X 0,Y 350.836,Z 370.191,A -85,B 0,C 180,E1 -14642.202,E2 -14642.202} C_VEL
LIN {X 0,Y 349.535,Z 383.725,A -85,B 0,C 180,E1 -14643.101,E2 -14643.101} C_VEL
LIN {X 0,Y 347.846,Z 397.471,A -85,B 0,C 180,E1 -14644.252,E2 -14644.252} C_VEL
LIN {X 0,Y 345.979,Z 410.042,A -85,B 0,C 180,E1 -14645.55,E2 -14645.55} C_VEL
LIN {X 0,Y 343.862,Z 422.701,A -85,B 0,C 180,E1 -14647.148,E2 -14647.148} C_VEL
LIN {X 0,Y 341.997,Z 434.134,A -85,B 0,C 180,E1 -14648.922,E2 -14648.922} C_VEL
LIN {X 0,Y 340.11,Z 443.76,A -85,B 0,C 180,E1 -14650.692,E2 -14650.692} C_VEL
LIN {X 0,Y 338.399,Z 452.2,A -85,B 0,C 180,E1 -14652.535,E2 -14652.535} C_VEL
LIN {X 0,Y 336.718,Z 460.959,A -85,B 0,C 180,E1 -14654.875,E2 -14654.875} C_VEL
LIN {X 0,Y 335.285,Z 468.215,A -85,B 0,C 180,E1 -14657.284,E2 -14657.284} C_VEL
LIN {X 0,Y 334.226,Z 473.957,A -85,B 0,C 180,E1 -14659.702,E2 -14659.702} C_VEL
LIN {X 0,Y 333.526,Z 478.227,A -85,B 0,C 180,E1 -14662.045,E2 -14662.045} C_VEL
LIN {X 0,Y 333.036,Z 480.794,A -85,B 0,C 180,E1 -14663.942,E2 -14663.942} C_VEL
LIN {X 0,Y 333.024,Z 482.058,A -85,B 0,C 180,E1 -14665.156,E2 -14665.156} C_VEL
LIN {X 0,Y 332.66,Z 483.776,A -85,B 0,C 180,E1 -14667.577,E2 -14667.577} C_VEL
LIN {X 0,Y 332.536,Z 484.371,A -85,B 0,C 180,E1 -14669.998,E2 -14669.998} C_VEL
LIN {X 0,Y 332.659,Z 483.815,A -85,B 0,C 180,E1 -14672.42,E2 -14672.42} C_VEL
LIN {X 0,Y 332.996,Z 482.153,A -85,B 0,C 180,E1 -14674.841,E2 -14674.841} C_VEL
LIN {X 0,Y 333.321,Z 479.371,A -85,B 0,C 180,E1 -14677.266,E2 -14677.266} C_VEL
LIN {X 0,Y 333.999,Z 475.372,A -85,B 0,C 180,E1 -14679.689,E2 -14679.689} C_VEL
LIN {X 0,Y 334.94,Z 470.051,A -85,B 0,C 180,E1 -14682.111,E2 -14682.111} C_VEL
LIN {X 0,Y 336.206,Z 463.257,A -85,B 0,C 180,E1 -14684.526,E2 -14684.526} C_VEL
LIN {X 0,Y 337.577,Z 456.357,A -85,B 0,C 180,E1 -14686.529,E2 -14686.529} C_VEL
LIN {X 0,Y 337.906,Z 454.662,A -85,B 0,C 180,E1 -14686.956,E2 -14686.956} C_VEL
LIN {X 0,Y 337.969,Z 451.44,A -85,B 0,C 180,E1 -14687.794,E2 -14687.794} C_VEL
LIN {X 0,Y 336.393,Z 446.129,A -85,B 0,C 180,E1 -14689.197,E2 -14689.197} C_VEL
LIN {X 0,Y 334.895,Z 440.413,A -85,B 0,C 180,E1 -14690.556,E2 -14690.556} C_VEL
LIN {X 0,Y 335.062,Z 436.506,A -85,B 0,C 180,E1 -14691.313,E2 -14691.313} C_VEL
LIN {X 0,Y 337.108,Z 425.049,A -85,B 0,C 180,E1 -14693.171,E2 -14693.171} C_VEL
LIN {X 0,Y 339.256,Z 412.752,A -85,B 0,C 180,E1 -14694.801,E2 -14694.801} C_VEL
LIN {X 0,Y 341.207,Z 400.632,A -85,B 0,C 180,E1 -14696.119,E2 -14696.119} C_VEL
LIN {X 0,Y 342.936,Z 387.529,A -85,B 0,C 180,E1 -14697.291,E2 -14697.291} C_VEL
LIN {X 0,Y 344.477,Z 372.995,A -85,B 0,C 180,E1 -14698.319,E2 -14698.319} C_VEL
LIN {X 0,Y 345.522,Z 359.181,A -85,B 0,C 180,E1 -14699.074,E2 -14699.074} C_VEL
LIN {X 0,Y 346.363,Z 344.468,A -85,B 0,C 180,E1 -14699.641,E2 -14699.641} C_VEL
LIN {X 0,Y 347.053,Z 322.116,A -85,B 0,C 180,E1 -14700.161,E2 -14700.161} C_VEL
LIN {X 0,Y 350.427,Z 211.074,A -85,B 0,C 180,E1 -14702.461,E2 -14702.461} C_VEL
LIN {X 0,Y 342.088,Z 193.653,A -85,B 0,C 180,E1 -14703.803,E2 -14703.803} C_VEL
LIN {X 0,Y 333.48,Z 177.681,A -85,B 0,C 180,E1 -14705.23,E2 -14705.23} C_VEL
LIN {X 0,Y 331.461,Z 174.009,A -85,B 0,C 180,E1 -14705.614,E2 -14705.614} C_VEL
LIN {X 0,Y 326.6,Z 161.419,A -85,B 0,C 180,E1 -14708.304,E2 -14708.304} C_VEL
LIN {X 0,Y 326.576,Z 161.418,A -85,B 0,C 180,E1 -14711.843,E2 -14711.843} C_VEL
LIN {X 0,Y 326.539,Z 161.431,A -85,B 0,C 180,E1 -14715.252,E2 -14715.252} C_VEL
LIN {X 0,Y 326.584,Z 161.428,A -85,B 0,C 180,E1 -14718.864,E2 -14718.864} C_VEL
LIN {X 0,Y 326.635,Z 161.413,A -85,B 0,C 180,E1 -14721.393,E2 -14721.393} C_VEL
LIN {X 0,Y 326.611,Z 161.415,A -85,B 0,C 180,E1 -14724.85,E2 -14724.85} C_VEL
LIN {X 0,Y 326.607,Z 161.428,A -85,B 0,C 180,E1 -14727.455,E2 -14727.455} C_VEL
LIN {X 0,Y 326.653,Z 161.403,A -85,B 0,C 180,E1 -14730.34,E2 -14730.34} C_VEL
LIN {X 0,Y 326.676,Z 161.417,A -85,B 0,C 180,E1 -14733.141,E2 -14733.141} C_VEL
LIN {X 0,Y 326.64,Z 161.407,A -85,B 0,C 180,E1 -14735.87,E2 -14735.87} C_VEL
LIN {X 0,Y 326.652,Z 161.409,A -85,B 0,C 180,E1 -14739.864,E2 -14739.864} C_VEL
LIN {X 0,Y 326.689,Z 161.407,A -85,B 0,C 180,E1 -14742.471,E2 -14742.471} C_VEL
LIN {X 0,Y 326.748,Z 161.391,A -85,B 0,C 180,E1 -14746.314,E2 -14746.314} C_VEL
LIN {X 0,Y 326.803,Z 161.401,A -85,B 0,C 180,E1 -14750.093,E2 -14750.093} C_VEL
LIN {X 0,Y 326.968,Z 161.362,A -85,B 0,C 180,E1 -14752.59,E2 -14752.59} C_VEL
LIN {X 0,Y 326.769,Z 161.394,A -85,B 0,C 180,E1 -14755.065,E2 -14755.065} C_VEL
LIN {X 0,Y 327.038,Z 161.37,A -85,B 0,C 180,E1 -14757.537,E2 -14757.537} C_VEL
LIN {X 0,Y 327.207,Z 161.327,A -85,B 0,C 180,E1 -14760,E2 -14760} C_VEL
LIN {X 0,Y 327.038,Z 161.366,A -85,B 0,C 180,E1 -14762.463,E2 -14762.463} C_VEL
LIN {X 0,Y 326.985,Z 161.357,A -85,B 0,C 180,E1 -14766.169,E2 -14766.169} C_VEL
LIN {X 0,Y 326.904,Z 161.378,A -85,B 0,C 180,E1 -14768.655,E2 -14768.655} C_VEL
LIN {X 0,Y 326.723,Z 161.389,A -85,B 0,C 180,E1 -14772.422,E2 -14772.422} C_VEL
LIN {X 0,Y 326.743,Z 161.4,A -85,B 0,C 180,E1 -14774.958,E2 -14774.958} C_VEL
LIN {X 0,Y 326.722,Z 161.389,A -85,B 0,C 180,E1 -14778.839,E2 -14778.839} C_VEL
LIN {X 0,Y 326.61,Z 161.419,A -85,B 0,C 180,E1 -14782.788,E2 -14782.788} C_VEL
LIN {X 0,Y 326.68,Z 161.405,A -85,B 0,C 180,E1 -14785.484,E2 -14785.484} C_VEL
LIN {X 0,Y 326.637,Z 161.407,A -85,B 0,C 180,E1 -14789.661,E2 -14789.661} C_VEL
LIN {X 0,Y 326.597,Z 161.416,A -85,B 0,C 180,E1 -14794.02,E2 -14794.02} C_VEL
LIN {X 0,Y 326.62,Z 161.423,A -85,B 0,C 180,E1 -14797.24,E2 -14797.24} C_VEL
LIN {X 0,Y 326.568,Z 161.387,A -85,B 0,C 180,E1 -14801.132,E2 -14801.132} C_VEL
LIN {X 0,Y 326.575,Z 161.431,A -85,B 0,C 180,E1 -14804.754,E2 -14804.754} C_VEL
LIN {X 0,Y 326.644,Z 161.601,A -85,B 0,C 180,E1 -14807.167,E2 -14807.167} C_VEL
LIN {X 0,Y 331.603,Z 178.386,A -85,B 0,C 180,E1 -14810.522,E2 -14810.522} C_VEL
LIN {X 0,Y 336.924,Z 196.854,A -85,B 0,C 180,E1 -14813.985,E2 -14813.985} C_VEL
LIN {X 0,Y 337.943,Z 200.35,A -85,B 0,C 180,E1 -14814.57,E2 -14814.57} C_VEL
LIN {X 0,Y 340.895,Z 208.335,A -85,B 0,C 180,E1 -14815.325,E2 -14815.325} C_VEL
LIN {X 0,Y 341.556,Z 217.557,A -85,B 0,C 180,E1 -14815.849,E2 -14815.849} C_VEL
LIN {X 0,Y 346.738,Z 263.551,A -85,B 0,C 180,E1 -14817.522,E2 -14817.522} C_VEL
LIN {X 0,Y 348.038,Z 276.557,A -85,B 0,C 180,E1 -14817.964,E2 -14817.964} C_VEL
LIN {X 0,Y 344.554,Z 391.498,A -85,B 0,C 180,E1 -14820.356,E2 -14820.356} C_VEL
LIN {X 0,Y 343.494,Z 406.367,A -85,B 0,C 180,E1 -14820.845,E2 -14820.845} C_VEL
LIN {X 0,Y 342.018,Z 421.021,A -85,B 0,C 180,E1 -14821.547,E2 -14821.547} C_VEL
LIN {X 0,Y 340.127,Z 435.348,A -85,B 0,C 180,E1 -14822.464,E2 -14822.464} C_VEL
LIN {X 0,Y 338.333,Z 447.829,A -85,B 0,C 180,E1 -14823.489,E2 -14823.489} C_VEL
LIN {X 0,Y 336.13,Z 460.759,A -85,B 0,C 180,E1 -14824.787,E2 -14824.787} C_VEL
LIN {X 0,Y 334.17,Z 471.741,A -85,B 0,C 180,E1 -14826.12,E2 -14826.12} C_VEL
LIN {X 0,Y 331.914,Z 483.99,A -85,B 0,C 180,E1 -14827.926,E2 -14827.926} C_VEL
LIN {X 0,Y 330.052,Z 494.679,A -85,B 0,C 180,E1 -14829.836,E2 -14829.836} C_VEL
LIN {X 0,Y 328.311,Z 504.383,A -85,B 0,C 180,E1 -14831.919,E2 -14831.919} C_VEL
LIN {X 0,Y 326.929,Z 512.768,A -85,B 0,C 180,E1 -14834.094,E2 -14834.094} C_VEL
LIN {X 0,Y 325.985,Z 519.731,A -85,B 0,C 180,E1 -14836.283,E2 -14836.283} C_VEL
LIN {X 0,Y 325.385,Z 526.211,A -85,B 0,C 180,E1 -14838.793,E2 -14838.793} C_VEL
LIN {X 0,Y 325.197,Z 531.239,A -85,B 0,C 180,E1 -14841.301,E2 -14841.301} C_VEL
LIN {X 0,Y 325.318,Z 534.938,A -85,B 0,C 180,E1 -14843.801,E2 -14843.801} C_VEL
LIN {X 0,Y 325.383,Z 537.371,A -85,B 0,C 180,E1 -14846.286,E2 -14846.286} C_VEL
LIN {X 0,Y 325.594,Z 538.607,A -85,B 0,C 180,E1 -14848.765,E2 -14848.765} C_VEL
LIN {X 0,Y 325.661,Z 538.771,A -85,B 0,C 180,E1 -14850.002,E2 -14850.002} C_VEL
LIN {X 0,Y 325.527,Z 538.137,A -85,B 0,C 180,E1 -14852.476,E2 -14852.476} C_VEL
LIN {X 0,Y 325.342,Z 536.295,A -85,B 0,C 180,E1 -14854.958,E2 -14854.958} C_VEL
LIN {X 0,Y 325.367,Z 534.584,A -85,B 0,C 180,E1 -14856.482,E2 -14856.482} C_VEL
LIN {X 0,Y 325.229,Z 531.207,A -85,B 0,C 180,E1 -14858.702,E2 -14858.702} C_VEL
LIN {X 0,Y 325.419,Z 526.166,A -85,B 0,C 180,E1 -14861.209,E2 -14861.209} C_VEL
LIN {X 0,Y 326.002,Z 519.679,A -85,B 0,C 180,E1 -14863.719,E2 -14863.719} C_VEL
LIN {X 0,Y 327.074,Z 511.56,A -85,B 0,C 180,E1 -14866.222,E2 -14866.222} C_VEL
LIN {X 0,Y 328.576,Z 502.932,A -85,B 0,C 180,E1 -14868.392,E2 -14868.392} C_VEL
LIN {X 0,Y 330.211,Z 493.401,A -85,B 0,C 180,E1 -14870.392,E2 -14870.392} C_VEL
LIN {X 0,Y 331.896,Z 483.865,A -85,B 0,C 180,E1 -14872.079,E2 -14872.079} C_VEL
LIN {X 0,Y 334.205,Z 471.583,A -85,B 0,C 180,E1 -14873.881,E2 -14873.881} C_VEL
LIN {X 0,Y 336.102,Z 460.569,A -85,B 0,C 180,E1 -14875.218,E2 -14875.218} C_VEL
LIN {X 0,Y 338.282,Z 447.528,A -85,B 0,C 180,E1 -14876.526,E2 -14876.526} C_VEL
LIN {X 0,Y 340.235,Z 436.319,A -85,B 0,C 180,E1 -14877.53,E2 -14877.53} C_VEL
LIN {X 0,Y 342.794,Z 423.47,A -85,B 0,C 180,E1 -14878.637,E2 -14878.637} C_VEL
LIN {X 0,Y 345.535,Z 408.633,A -85,B 0,C 180,E1 -14879.638,E2 -14879.638} C_VEL
LIN {X 0,Y 348.129,Z 391.641,A -85,B 0,C 180,E1 -14880.522,E2 -14880.522} C_VEL
LIN {X 0,Y 349.966,Z 375.206,A -85,B 0,C 180,E1 -14881.14,E2 -14881.14} C_VEL
LIN {X 0,Y 355.891,Z 312.693,A -85,B 0,C 180,E1 -14883.189,E2 -14883.189} C_VEL
LIN {X 0,Y 359.601,Z 277.96,A -85,B 0,C 180,E1 -14884.402,E2 -14884.402} C_VEL
LIN {X 0,Y 359.676,Z 262.824,A -85,B 0,C 180,E1 -14885.31,E2 -14885.31} C_VEL
LIN {X 0,Y 359.056,Z 248.515,A -85,B 0,C 180,E1 -14886.421,E2 -14886.421} C_VEL
LIN {X 0,Y 358.13,Z 234.644,A -85,B 0,C 180,E1 -14887.704,E2 -14887.704} C_VEL
LIN {X 0,Y 357.855,Z 232.75,A -85,B 0,C 180,E1 -14887.938,E2 -14887.938} C_VEL
LIN {X 0,Y 355.057,Z 226.926,A -85,B 0,C 180,E1 -14889.469,E2 -14889.469} C_VEL
LIN {X 0,Y 353.903,Z 222.042,A -85,B 0,C 180,E1 -14891.868,E2 -14891.868} C_VEL
LIN {X 0,Y 352.707,Z 218.954,A -85,B 0,C 180,E1 -14894.221,E2 -14894.221} C_VEL
LIN {X 0,Y 352.06,Z 217.466,A -85,B 0,C 180,E1 -14895.945,E2 -14895.945} C_VEL
LIN {X 0,Y 351.605,Z 216.605,A -85,B 0,C 180,E1 -14897.696,E2 -14897.696} C_VEL
LIN {X 0,Y 351.172,Z 216.574,A -85,B 0,C 180,E1 -14900.177,E2 -14900.177} C_VEL
LIN {X 0,Y 351.007,Z 217.194,A -85,B 0,C 180,E1 -14901.633,E2 -14901.633} C_VEL
LIN {X 0,Y 350.998,Z 219.124,A -85,B 0,C 180,E1 -14904.051,E2 -14904.051} C_VEL
LIN {X 0,Y 354.315,Z 224.49,A -85,B 0,C 180,E1 -14906.358,E2 -14906.358} C_VEL
LIN {X 0,Y 356.959,Z 229.36,A -85,B 0,C 180,E1 -14907.846,E2 -14907.846} C_VEL
LIN {X 0,Y 359.457,Z 234.309,A -85,B 0,C 180,E1 -14909.084,E2 -14909.084} C_VEL
LIN {X 0,Y 360.479,Z 236.782,A -85,B 0,C 180,E1 -14909.574,E2 -14909.574} C_VEL
LIN {X 0,Y 362.12,Z 247.966,A -85,B 0,C 180,E1 -14910.892,E2 -14910.892} C_VEL
LIN {X 0,Y 362.2,Z 249.475,A -85,B 0,C 180,E1 -14911.025,E2 -14911.025} C_VEL
LIN {X 0,Y 351.663,Z 327.414,A -85,B 0,C 180,E1 -14914.236,E2 -14914.236} C_VEL
LIN {X 0,Y 349.843,Z 345.436,A -85,B 0,C 180,E1 -14915.125,E2 -14915.125} C_VEL
LIN {X 0,Y 348.135,Z 359.192,A -85,B 0,C 180,E1 -14916.033,E2 -14916.033} C_VEL
LIN {X 0,Y 345.877,Z 373.999,A -85,B 0,C 180,E1 -14917.29,E2 -14917.29} C_VEL
LIN {X 0,Y 343.536,Z 387.013,A -85,B 0,C 180,E1 -14918.708,E2 -14918.708} C_VEL
LIN {X 0,Y 341.441,Z 397.67,A -85,B 0,C 180,E1 -14920.146,E2 -14920.146} C_VEL
LIN {X 0,Y 339.428,Z 406.562,A -85,B 0,C 180,E1 -14921.594,E2 -14921.594} C_VEL
LIN {X 0,Y 337.285,Z 415.515,A -85,B 0,C 180,E1 -14923.382,E2 -14923.382} C_VEL
LIN {X 0,Y 335.285,Z 422.669,A -85,B 0,C 180,E1 -14925.118,E2 -14925.118} C_VEL
LIN {X 0,Y 333.316,Z 429.424,A -85,B 0,C 180,E1 -14927.209,E2 -14927.209} C_VEL
LIN {X 0,Y 331.725,Z 433.933,A -85,B 0,C 180,E1 -14929.008,E2 -14929.008} C_VEL
LIN {X 0,Y 330.905,Z 436.28,A -85,B 0,C 180,E1 -14930.218,E2 -14930.218} C_VEL
LIN {X 0,Y 330.065,Z 438.207,A -85,B 0,C 180,E1 -14931.428,E2 -14931.428} C_VEL
LIN {X 0,Y 329.384,Z 439.698,A -85,B 0,C 180,E1 -14932.645,E2 -14932.645} C_VEL
LIN {X 0,Y 328.84,Z 440.729,A -85,B 0,C 180,E1 -14933.866,E2 -14933.866} C_VEL
LIN {X 0,Y 328.398,Z 441.313,A -85,B 0,C 180,E1 -14935.089,E2 -14935.089} C_VEL
LIN {X 0,Y 327.919,Z 441.521,A -85,B 0,C 180,E1 -14936.314,E2 -14936.314} C_VEL
LIN {X 0,Y 327.618,Z 441.299,A -85,B 0,C 180,E1 -14937.541,E2 -14937.541} C_VEL
LIN {X 0,Y 327.247,Z 440.678,A -85,B 0,C 180,E1 -14938.77,E2 -14938.77} C_VEL
LIN {X 0,Y 326.945,Z 439.601,A -85,B 0,C 180,E1 -14940,E2 -14940} C_VEL
LIN {X 0,Y 326.958,Z 438.078,A -85,B 0,C 180,E1 -14941.232,E2 -14941.232} C_VEL
LIN {X 0,Y 326.831,Z 435.006,A -85,B 0,C 180,E1 -14943.082,E2 -14943.082} C_VEL
LIN {X 0,Y 326.722,Z 430.898,A -85,B 0,C 180,E1 -14944.936,E2 -14944.936} C_VEL
LIN {X 0,Y 327.127,Z 424.648,A -85,B 0,C 180,E1 -14947.096,E2 -14947.096} C_VEL
LIN {X 0,Y 327.483,Z 416.982,A -85,B 0,C 180,E1 -14949.174,E2 -14949.174} C_VEL
LIN {X 0,Y 328.045,Z 408.047,A -85,B 0,C 180,E1 -14951.117,E2 -14951.117} C_VEL
LIN {X 0,Y 328.611,Z 399.444,A -85,B 0,C 180,E1 -14952.663,E2 -14952.663} C_VEL
LIN {X 0,Y 329.23,Z 389.143,A -85,B 0,C 180,E1 -14954.211,E2 -14954.211} C_VEL
LIN {X 0,Y 330.084,Z 376.53,A -85,B 0,C 180,E1 -14955.752,E2 -14955.752} C_VEL
LIN {X 0,Y 330.759,Z 363.643,A -85,B 0,C 180,E1 -14957.024,E2 -14957.024} C_VEL
LIN {X 0,Y 331.528,Z 349.118,A -85,B 0,C 180,E1 -14958.141,E2 -14958.141} C_VEL
LIN {X 0,Y 331.978,Z 334.296,A -85,B 0,C 180,E1 -14958.995,E2 -14958.995} C_VEL
LIN {X 0,Y 332.462,Z 319.937,A -85,B 0,C 180,E1 -14959.568,E2 -14959.568} C_VEL
LIN {X 0,Y 335.569,Z 229.714,A -85,B 0,C 180,E1 -14962.352,E2 -14962.352} C_VEL
LIN {X 0,Y 331.84,Z 204.052,A -85,B 0,C 180,E1 -14963.406,E2 -14963.406} C_VEL
LIN {X 0,Y 333.107,Z 192.151,A -85,B 0,C 180,E1 -14965.963,E2 -14965.963} C_VEL
LIN {X 0,Y 332.725,Z 188.182,A -85,B 0,C 180,E1 -14966.876,E2 -14966.876} C_VEL
LIN {X 0,Y 329.845,Z 175.23,A -85,B 0,C 180,E1 -14970.047,E2 -14970.047} C_VEL
LIN {X 0,Y 326.633,Z 161.424,A -85,B 0,C 180,E1 -14973.591,E2 -14973.591} C_VEL
LIN {X 0,Y 326.629,Z 161.425,A -85,B 0,C 180,E1 -14977.237,E2 -14977.237} C_VEL
LIN {X 0,Y 326.58,Z 161.424,A -85,B 0,C 180,E1 -14981.13,E2 -14981.13} C_VEL
LIN {X 0,Y 326.561,Z 161.427,A -85,B 0,C 180,E1 -14984.747,E2 -14984.747} C_VEL
LIN {X 0,Y 326.582,Z 161.429,A -85,B 0,C 180,E1 -14988.154,E2 -14988.154} C_VEL
LIN {X 0,Y 326.602,Z 161.461,A -85,B 0,C 180,E1 -14991.848,E2 -14991.848} C_VEL
LIN {X 0,Y 331.736,Z 174.622,A -85,B 0,C 180,E1 -14994.592,E2 -14994.592} C_VEL
LIN {X 0,Y 342.228,Z 193.897,A -85,B 0,C 180,E1 -14996.335,E2 -14996.335} C_VEL
LIN {X 0,Y 349.668,Z 209.55,A -85,B 0,C 180,E1 -14997.535,E2 -14997.535} C_VEL
LIN {X 0,Y 350.385,Z 211.178,A -85,B 0,C 180,E1 -14997.65,E2 -14997.65} C_VEL
LIN {X 0,Y 348.047,Z 287.33,A -85,B 0,C 180,E1 -14999.226,E2 -14999.226} C_VEL
LIN {X 0,Y 346.353,Z 342.118,A -85,B 0,C 180,E1 -15000.397,E2 -15000.397} C_VEL
LIN {X 0,Y 345.545,Z 357.664,A -85,B 0,C 180,E1 -15000.967,E2 -15000.967} C_VEL
LIN {X 0,Y 344.463,Z 372.31,A -85,B 0,C 180,E1 -15001.746,E2 -15001.746} C_VEL
LIN {X 0,Y 343.066,Z 386.202,A -85,B 0,C 180,E1 -15002.717,E2 -15002.717} C_VEL
LIN {X 0,Y 341.288,Z 399.571,A -85,B 0,C 180,E1 -15003.884,E2 -15003.884} C_VEL
LIN {X 0,Y 339.33,Z 411.87,A -85,B 0,C 180,E1 -15005.202,E2 -15005.202} C_VEL
LIN {X 0,Y 337.192,Z 424.314,A -85,B 0,C 180,E1 -15006.832,E2 -15006.832} C_VEL
LIN {X 0,Y 335.403,Z 434.715,A -85,B 0,C 180,E1 -15008.487,E2 -15008.487} C_VEL
LIN {X 0,Y 333.432,Z 444.343,A -85,B 0,C 180,E1 -15010.29,E2 -15010.29} C_VEL
LIN {X 0,Y 331.43,Z 453.741,A -85,B 0,C 180,E1 -15012.41,E2 -15012.41} C_VEL
LIN {X 0,Y 329.88,Z 461.544,A -85,B 0,C 180,E1 -15014.554,E2 -15014.554} C_VEL
LIN {X 0,Y 328.374,Z 468.8,A -85,B 0,C 180,E1 -15017.012,E2 -15017.012} C_VEL
LIN {X 0,Y 327.248,Z 474.544,A -85,B 0,C 180,E1 -15019.48,E2 -15019.48} C_VEL
LIN {X 0,Y 326.483,Z 478.974,A -85,B 0,C 180,E1 -15021.979,E2 -15021.979} C_VEL
LIN {X 0,Y 325.994,Z 481.38,A -85,B 0,C 180,E1 -15023.81,E2 -15023.81} C_VEL
LIN {X 0,Y 325.793,Z 483.639,A -85,B 0,C 180,E1 -15026.288,E2 -15026.288} C_VEL
LIN {X 0,Y 325.491,Z 484.803,A -85,B 0,C 180,E1 -15028.761,E2 -15028.761} C_VEL
LIN {X 0,Y 325.491,Z 484.816,A -85,B 0,C 180,E1 -15031.236,E2 -15031.236} C_VEL
LIN {X 0,Y 325.789,Z 483.703,A -85,B 0,C 180,E1 -15033.709,E2 -15033.709} C_VEL
LIN {X 0,Y 325.984,Z 481.501,A -85,B 0,C 180,E1 -15036.187,E2 -15036.187} C_VEL
LIN {X 0,Y 326.624,Z 478.113,A -85,B 0,C 180,E1 -15038.661,E2 -15038.661} C_VEL
LIN {X 0,Y 327.513,Z 473.466,A -85,B 0,C 180,E1 -15041.134,E2 -15041.134} C_VEL
LIN {X 0,Y 328.658,Z 467.43,A -85,B 0,C 180,E1 -15043.603,E2 -15043.603} C_VEL
LIN {X 0,Y 330.095,Z 460.891,A -85,B 0,C 180,E1 -15045.749,E2 -15045.749} C_VEL
LIN {X 0,Y 331.643,Z 452.97,A -85,B 0,C 180,E1 -15047.893,E2 -15047.893} C_VEL
LIN {X 0,Y 333.657,Z 443.414,A -85,B 0,C 180,E1 -15050.014,E2 -15050.014} C_VEL
LIN {X 0,Y 335.062,Z 436.506,A -85,B 0,C 180,E1 -15051.313,E2 -15051.313} C_VEL
LIN {X 0,Y 335.253,Z 432.497,A -85,B 0,C 180,E1 -15052.058,E2 -15052.058} C_VEL
LIN {X 0,Y 333.819,Z 426.002,A -85,B 0,C 180,E1 -15053.319,E2 -15053.319} C_VEL
LIN {X 0,Y 332.439,Z 419.165,A -85,B 0,C 180,E1 -15054.527,E2 -15054.527} C_VEL
LIN {X 0,Y 332.641,Z 414.571,A -85,B 0,C 180,E1 -15055.161,E2 -15055.161} C_VEL
LIN {X 0,Y 334.882,Z 401.196,A -85,B 0,C 180,E1 -15056.651,E2 -15056.651} C_VEL
LIN {X 0,Y 336.676,Z 388.085,A -85,B 0,C 180,E1 -15057.842,E2 -15057.842} C_VEL
LIN {X 0,Y 338.259,Z 373.82,A -85,B 0,C 180,E1 -15058.869,E2 -15058.869} C_VEL
LIN {X 0,Y 339.38,Z 359.572,A -85,B 0,C 180,E1 -15059.66,E2 -15059.66} C_VEL
LIN {X 0,Y 340.228,Z 344.968,A -85,B 0,C 180,E1 -15060.23,E2 -15060.23} C_VEL
LIN {X 0,Y 341.05,Z 319.008,A -85,B 0,C 180,E1 -15060.835,E2 -15060.835} C_VEL
LIN {X 0,Y 344.45,Z 213.279,A -85,B 0,C 180,E1 -15063.052,E2 -15063.052} C_VEL
LIN {X 0,Y 335.524,Z 194.748,A -85,B 0,C 180,E1 -15064.541,E2 -15064.541} C_VEL
LIN {X 0,Y 326.366,Z 178.033,A -85,B 0,C 180,E1 -15066.122,E2 -15066.122} C_VEL
LIN {X 0,Y 324.394,Z 174.661,A -85,B 0,C 180,E1 -15066.506,E2 -15066.506} C_VEL
LIN {X 0,Y 319.57,Z 162.278,A -85,B 0,C 180,E1 -15069.225,E2 -15069.225} C_VEL
LIN {X 0,Y 319.558,Z 162.307,A -85,B 0,C 180,E1 -15072.98,E2 -15072.98} C_VEL
LIN {X 0,Y 319.571,Z 162.296,A -85,B 0,C 180,E1 -15077.019,E2 -15077.019} C_VEL
LIN {X 0,Y 319.574,Z 162.296,A -85,B 0,C 180,E1 -15080.375,E2 -15080.375} C_VEL
LIN {X 0,Y 319.551,Z 162.305,A -85,B 0,C 180,E1 -15083.571,E2 -15083.571} C_VEL
LIN {X 0,Y 319.57,Z 162.298,A -85,B 0,C 180,E1 -15086.685,E2 -15086.685} C_VEL
LIN {X 0,Y 319.585,Z 162.284,A -85,B 0,C 180,E1 -15089.616,E2 -15089.616} C_VEL
LIN {X 0,Y 319.608,Z 162.298,A -85,B 0,C 180,E1 -15092.498,E2 -15092.498} C_VEL
LIN {X 0,Y 319.594,Z 162.282,A -85,B 0,C 180,E1 -15095.303,E2 -15095.303} C_VEL
LIN {X 0,Y 319.586,Z 162.3,A -85,B 0,C 180,E1 -15098.047,E2 -15098.047} C_VEL
LIN {X 0,Y 319.679,Z 162.269,A -85,B 0,C 180,E1 -15100.962,E2 -15100.962} C_VEL
LIN {X 0,Y 319.72,Z 162.277,A -85,B 0,C 180,E1 -15105.275,E2 -15105.275} C_VEL
LIN {X 0,Y 319.747,Z 162.28,A -85,B 0,C 180,E1 -15109.872,E2 -15109.872} C_VEL
LIN {X 0,Y 319.922,Z 162.241,A -85,B 0,C 180,E1 -15112.426,E2 -15112.426} C_VEL
LIN {X 0,Y 319.738,Z 162.268,A -85,B 0,C 180,E1 -15114.956,E2 -15114.956} C_VEL
LIN {X 0,Y 319.981,Z 162.249,A -85,B 0,C 180,E1 -15117.482,E2 -15117.482} C_VEL
LIN {X 0,Y 320.159,Z 162.205,A -85,B 0,C 180,E1 -15120,E2 -15120} C_VEL
LIN {X 0,Y 319.982,Z 162.245,A -85,B 0,C 180,E1 -15122.518,E2 -15122.518} C_VEL
LIN {X 0,Y 319.941,Z 162.232,A -85,B 0,C 180,E1 -15126.306,E2 -15126.306} C_VEL
LIN {X 0,Y 319.832,Z 162.261,A -85,B 0,C 180,E1 -15128.848,E2 -15128.848} C_VEL
LIN {X 0,Y 319.67,Z 162.265,A -85,B 0,C 180,E1 -15132.7,E2 -15132.7} C_VEL
LIN {X 0,Y 319.689,Z 162.282,A -85,B 0,C 180,E1 -15135.296,E2 -15135.296} C_VEL
LIN {X 0,Y 319.663,Z 162.268,A -85,B 0,C 180,E1 -15139.256,E2 -15139.256} C_VEL
LIN {X 0,Y 319.56,Z 162.294,A -85,B 0,C 180,E1 -15143.32,E2 -15143.32} C_VEL
LIN {X 0,Y 319.624,Z 162.289,A -85,B 0,C 180,E1 -15146.089,E2 -15146.089} C_VEL
LIN {X 0,Y 319.569,Z 162.29,A -85,B 0,C 180,E1 -15148.935,E2 -15148.935} C_VEL
LIN {X 0,Y 319.521,Z 162.309,A -85,B 0,C 180,E1 -15151.863,E2 -15151.863} C_VEL
LIN {X 0,Y 319.571,Z 162.299,A -85,B 0,C 180,E1 -15155.544,E2 -15155.544} C_VEL
LIN {X 0,Y 319.565,Z 162.286,A -85,B 0,C 180,E1 -15158.009,E2 -15158.009} C_VEL
LIN {X 0,Y 319.517,Z 162.27,A -85,B 0,C 180,E1 -15161.598,E2 -15161.598} C_VEL
LIN {X 0,Y 319.563,Z 162.305,A -85,B 0,C 180,E1 -15165.273,E2 -15165.273} C_VEL
LIN {X 0,Y 319.592,Z 162.463,A -85,B 0,C 180,E1 -15166.624,E2 -15166.624} C_VEL
LIN {X 0,Y 324.728,Z 179.914,A -85,B 0,C 180,E1 -15170.203,E2 -15170.203} C_VEL
LIN {X 0,Y 329.53,Z 196.49,A -85,B 0,C 180,E1 -15173.335,E2 -15173.335} C_VEL
LIN {X 0,Y 335.026,Z 210.931,A -85,B 0,C 180,E1 -15174.795,E2 -15174.795} C_VEL
LIN {X 0,Y 335.416,Z 216.895,A -85,B 0,C 180,E1 -15175.129,E2 -15175.129} C_VEL
LIN {X 0,Y 340.411,Z 261.377,A -85,B 0,C 180,E1 -15176.8,E2 -15176.8} C_VEL
LIN {X 0,Y 341.994,Z 277.603,A -85,B 0,C 180,E1 -15177.365,E2 -15177.365} C_VEL
LIN {X 0,Y 338.384,Z 391.013,A -85,B 0,C 180,E1 -15179.76,E2 -15179.76} C_VEL
LIN {X 0,Y 337.317,Z 405.84,A -85,B 0,C 180,E1 -15180.258,E2 -15180.258} C_VEL
LIN {X 0,Y 335.769,Z 420.471,A -85,B 0,C 180,E1 -15180.967,E2 -15180.967} C_VEL
LIN {X 0,Y 333.825,Z 434.787,A -85,B 0,C 180,E1 -15181.899,E2 -15181.899} C_VEL
LIN {X 0,Y 332.044,Z 446.638,A -85,B 0,C 180,E1 -15182.88,E2 -15182.88} C_VEL
LIN {X 0,Y 329.911,Z 458.888,A -85,B 0,C 180,E1 -15184.108,E2 -15184.108} C_VEL
LIN {X 0,Y 327.587,Z 471.157,A -85,B 0,C 180,E1 -15185.609,E2 -15185.609} C_VEL
LIN {X 0,Y 325.269,Z 483.405,A -85,B 0,C 180,E1 -15187.45,E2 -15187.45} C_VEL
LIN {X 0,Y 323.311,Z 493.751,A -85,B 0,C 180,E1 -15189.325,E2 -15189.325} C_VEL
LIN {X 0,Y 321.475,Z 503.794,A -85,B 0,C 180,E1 -15191.521,E2 -15191.521} C_VEL
LIN {X 0,Y 319.978,Z 512.174,A -85,B 0,C 180,E1 -15193.739,E2 -15193.739} C_VEL
LIN {X 0,Y 319.015,Z 519.141,A -85,B 0,C 180,E1 -15195.977,E2 -15195.977} C_VEL
LIN {X 0,Y 318.346,Z 525.62,A -85,B 0,C 180,E1 -15198.541,E2 -15198.541} C_VEL
LIN {X 0,Y 318.099,Z 530.646,A -85,B 0,C 180,E1 -15201.105,E2 -15201.105} C_VEL
LIN {X 0,Y 318.244,Z 534.35,A -85,B 0,C 180,E1 -15203.662,E2 -15203.662} C_VEL
LIN {X 0,Y 318.292,Z 536.784,A -85,B 0,C 180,E1 -15206.204,E2 -15206.204} C_VEL
LIN {X 0,Y 318.457,Z 537.557,A -85,B 0,C 180,E1 -15207.472,E2 -15207.472} C_VEL
LIN {X 0,Y 318.612,Z 538.189,A -85,B 0,C 180,E1 -15210.002,E2 -15210.002} C_VEL
LIN {X 0,Y 318.458,Z 537.552,A -85,B 0,C 180,E1 -15212.531,E2 -15212.531} C_VEL
LIN {X 0,Y 318.277,Z 535.709,A -85,B 0,C 180,E1 -15215.069,E2 -15215.069} C_VEL
LIN {X 0,Y 318.295,Z 534.166,A -85,B 0,C 180,E1 -15216.483,E2 -15216.483} C_VEL
LIN {X 0,Y 318.133,Z 530.613,A -85,B 0,C 180,E1 -15218.897,E2 -15218.897} C_VEL
LIN {X 0,Y 318.382,Z 525.573,A -85,B 0,C 180,E1 -15221.461,E2 -15221.461} C_VEL
LIN {X 0,Y 319.007,Z 519.084,A -85,B 0,C 180,E1 -15224.026,E2 -15224.026} C_VEL
LIN {X 0,Y 320.181,Z 510.967,A -85,B 0,C 180,E1 -15226.581,E2 -15226.581} C_VEL
LIN {X 0,Y 321.743,Z 502.338,A -85,B 0,C 180,E1 -15228.797,E2 -15228.797} C_VEL
LIN {X 0,Y 323.456,Z 492.566,A -85,B 0,C 180,E1 -15230.886,E2 -15230.886} C_VEL
LIN {X 0,Y 325.592,Z 481.347,A -85,B 0,C 180,E1 -15232.865,E2 -15232.865} C_VEL
LIN {X 0,Y 327.832,Z 469.829,A -85,B 0,C 180,E1 -15234.543,E2 -15234.543} C_VEL
LIN {X 0,Y 330.175,Z 457.328,A -85,B 0,C 180,E1 -15236.043,E2 -15236.043} C_VEL
LIN {X 0,Y 332.202,Z 445.738,A -85,B 0,C 180,E1 -15237.235,E2 -15237.235} C_VEL
LIN {X 0,Y 335.328,Z 431.814,A -85,B 0,C 180,E1 -15238.649,E2 -15238.649} C_VEL
LIN {X 0,Y 338.536,Z 416.668,A -85,B 0,C 180,E1 -15239.885,E2 -15239.885} C_VEL
LIN {X 0,Y 341.544,Z 400.558,A -85,B 0,C 180,E1 -15240.875,E2 -15240.875} C_VEL
LIN {X 0,Y 344.048,Z 382.991,A -85,B 0,C 180,E1 -15241.694,E2 -15241.694} C_VEL
LIN {X 0,Y 351.428,Z 312.442,A -85,B 0,C 180,E1 -15244.098,E2 -15244.098} C_VEL
LIN {X 0,Y 355.303,Z 279.145,A -85,B 0,C 180,E1 -15245.291,E2 -15245.291} C_VEL
LIN {X 0,Y 355.558,Z 265.195,A -85,B 0,C 180,E1 -15246.16,E2 -15246.16} C_VEL
LIN {X 0,Y 355.182,Z 250.897,A -85,B 0,C 180,E1 -15247.306,E2 -15247.306} C_VEL
LIN {X 0,Y 354.612,Z 237.98,A -85,B 0,C 180,E1 -15248.546,E2 -15248.546} C_VEL
LIN {X 0,Y 352.003,Z 232.467,A -85,B 0,C 180,E1 -15250.049,E2 -15250.049} C_VEL
LIN {X 0,Y 348.776,Z 226.519,A -85,B 0,C 180,E1 -15252.365,E2 -15252.365} C_VEL
LIN {X 0,Y 347.859,Z 224.812,A -85,B 0,C 180,E1 -15253.388,E2 -15253.388} C_VEL
LIN {X 0,Y 347.122,Z 222.978,A -85,B 0,C 180,E1 -15255.125,E2 -15255.125} C_VEL
LIN {X 0,Y 346.595,Z 221.772,A -85,B 0,C 180,E1 -15256.886,E2 -15256.886} C_VEL
LIN {X 0,Y 346.081,Z 221.262,A -85,B 0,C 180,E1 -15259.471,E2 -15259.471} C_VEL
LIN {X 0,Y 346.052,Z 221.637,A -85,B 0,C 180,E1 -15260.42,E2 -15260.42} C_VEL
LIN {X 0,Y 348.038,Z 224.763,A -85,B 0,C 180,E1 -15263.145,E2 -15263.145} C_VEL
LIN {X 0,Y 349.132,Z 226.482,A -85,B 0,C 180,E1 -15264.145,E2 -15264.145} C_VEL
LIN {X 0,Y 351.8,Z 230.882,A -85,B 0,C 180,E1 -15266.051,E2 -15266.051} C_VEL
LIN {X 0,Y 354.32,Z 235.845,A -85,B 0,C 180,E1 -15267.581,E2 -15267.581} C_VEL
LIN {X 0,Y 356.794,Z 241.118,A -85,B 0,C 180,E1 -15268.892,E2 -15268.892} C_VEL
LIN {X 0,Y 358.084,Z 251.184,A -85,B 0,C 180,E1 -15270.116,E2 -15270.116} C_VEL
LIN {X 0,Y 346.769,Z 329.905,A -85,B 0,C 180,E1 -15273.448,E2 -15273.448} C_VEL
LIN {X 0,Y 345.084,Z 345.183,A -85,B 0,C 180,E1 -15274.219,E2 -15274.219} C_VEL
LIN {X 0,Y 343.365,Z 358.559,A -85,B 0,C 180,E1 -15275.095,E2 -15275.095} C_VEL
LIN {X 0,Y 341.049,Z 372.944,A -85,B 0,C 180,E1 -15276.307,E2 -15276.307} C_VEL
LIN {X 0,Y 338.757,Z 385.128,A -85,B 0,C 180,E1 -15277.591,E2 -15277.591} C_VEL
LIN {X 0,Y 336.381,Z 396.198,A -85,B 0,C 180,E1 -15279.035,E2 -15279.035} C_VEL
LIN {X 0,Y 333.974,Z 406.321,A -85,B 0,C 180,E1 -15280.644,E2 -15280.644} C_VEL
LIN {X 0,Y 332.072,Z 413.983,A -85,B 0,C 180,E1 -15282.13,E2 -15282.13} C_VEL
LIN {X 0,Y 329.85,Z 421.721,A -85,B 0,C 180,E1 -15283.92,E2 -15283.92} C_VEL
LIN {X 0,Y 327.856,Z 428.002,A -85,B 0,C 180,E1 -15285.729,E2 -15285.729} C_VEL
LIN {X 0,Y 326.102,Z 433.044,A -85,B 0,C 180,E1 -15287.554,E2 -15287.554} C_VEL
LIN {X 0,Y 324.589,Z 436.965,A -85,B 0,C 180,E1 -15289.395,E2 -15289.395} C_VEL
LIN {X 0,Y 323.25,Z 439.837,A -85,B 0,C 180,E1 -15291.246,E2 -15291.246} C_VEL
LIN {X 0,Y 322.517,Z 441.197,A -85,B 0,C 180,E1 -15292.487,E2 -15292.487} C_VEL
LIN {X 0,Y 321.927,Z 442.103,A -85,B 0,C 180,E1 -15293.734,E2 -15293.734} C_VEL
LIN {X 0,Y 321.469,Z 442.6,A -85,B 0,C 180,E1 -15294.983,E2 -15294.983} C_VEL
LIN {X 0,Y 320.956,Z 442.719,A -85,B 0,C 180,E1 -15296.234,E2 -15296.234} C_VEL
LIN {X 0,Y 320.617,Z 442.401,A -85,B 0,C 180,E1 -15297.487,E2 -15297.487} C_VEL
LIN {X 0,Y 320.231,Z 441.647,A -85,B 0,C 180,E1 -15298.743,E2 -15298.743} C_VEL
LIN {X 0,Y 319.918,Z 440.48,A -85,B 0,C 180,E1 -15300,E2 -15300} C_VEL
LIN {X 0,Y 319.832,Z 437.904,A -85,B 0,C 180,E1 -15301.889,E2 -15301.889} C_VEL
LIN {X 0,Y 319.694,Z 434.343,A -85,B 0,C 180,E1 -15303.782,E2 -15303.782} C_VEL
LIN {X 0,Y 319.851,Z 429.684,A -85,B 0,C 180,E1 -15305.675,E2 -15305.675} C_VEL
LIN {X 0,Y 320.179,Z 422.752,A -85,B 0,C 180,E1 -15307.885,E2 -15307.885} C_VEL
LIN {X 0,Y 320.528,Z 415.231,A -85,B 0,C 180,E1 -15309.804,E2 -15309.804} C_VEL
LIN {X 0,Y 321.151,Z 406.178,A -85,B 0,C 180,E1 -15311.679,E2 -15311.679} C_VEL
LIN {X 0,Y 321.874,Z 395.006,A -85,B 0,C 180,E1 -15313.575,E2 -15313.575} C_VEL
LIN {X 0,Y 322.61,Z 383.506,A -85,B 0,C 180,E1 -15315.154,E2 -15315.154} C_VEL
LIN {X 0,Y 323.476,Z 370.562,A -85,B 0,C 180,E1 -15316.603,E2 -15316.603} C_VEL
LIN {X 0,Y 324.199,Z 356.632,A -85,B 0,C 180,E1 -15317.831,E2 -15317.831} C_VEL
LIN {X 0,Y 324.811,Z 342.86,A -85,B 0,C 180,E1 -15318.775,E2 -15318.775} C_VEL
LIN {X 0,Y 325.272,Z 328.771,A -85,B 0,C 180,E1 -15319.485,E2 -15319.485} C_VEL
LIN {X 0,Y 326.213,Z 297.391,A -85,B 0,C 180,E1 -15320.534,E2 -15320.534} C_VEL
LIN {X 0,Y 328.762,Z 230.765,A -85,B 0,C 180,E1 -15322.654,E2 -15322.654} C_VEL
LIN {X 0,Y 325.003,Z 204.393,A -85,B 0,C 180,E1 -15323.75,E2 -15323.75} C_VEL
LIN {X 0,Y 326.202,Z 193.131,A -85,B 0,C 180,E1 -15326.211,E2 -15326.211} C_VEL
LIN {X 0,Y 325.461,Z 188.092,A -85,B 0,C 180,E1 -15327.407,E2 -15327.407} C_VEL
LIN {X 0,Y 322.808,Z 176.087,A -85,B 0,C 180,E1 -15330.41,E2 -15330.41} C_VEL
LIN {X 0,Y 319.585,Z 162.303,A -85,B 0,C 180,E1 -15334.004,E2 -15334.004} C_VEL
LIN {X 0,Y 319.554,Z 162.307,A -85,B 0,C 180,E1 -15337.648,E2 -15337.648} C_VEL
LIN {X 0,Y 319.531,Z 162.304,A -85,B 0,C 180,E1 -15341.288,E2 -15341.288} C_VEL
LIN {X 0,Y 319.52,Z 162.304,A -85,B 0,C 180,E1 -15344.737,E2 -15344.737} C_VEL
LIN {X 0,Y 319.567,Z 162.296,A -85,B 0,C 180,E1 -15347.017,E2 -15347.017} C_VEL
LIN {X 0,Y 319.593,Z 162.306,A -85,B 0,C 180,E1 -15350.927,E2 -15350.927} C_VEL
LIN {X 0,Y 319.953,Z 163.862,A -85,B 0,C 180,E1 -15351.24,E2 -15351.24} C_VEL
LIN {X 0,Y 323.945,Z 173.571,A -85,B 0,C 180,E1 -15353.39,E2 -15353.39} C_VEL
LIN {X 0,Y 324.698,Z 175.304,A -85,B 0,C 180,E1 -15353.707,E2 -15353.707} C_VEL
LIN {X 0,Y 333.437,Z 190.773,A -85,B 0,C 180,E1 -15355.223,E2 -15355.223} C_VEL
LIN {X 0,Y 342.347,Z 208.661,A -85,B 0,C 180,E1 -15356.716,E2 -15356.716} C_VEL
LIN {X 0,Y 344.402,Z 213.341,A -85,B 0,C 180,E1 -15357.059,E2 -15357.059} C_VEL
LIN {X 0,Y 341.954,Z 288.454,A -85,B 0,C 180,E1 -15358.631,E2 -15358.631} C_VEL
LIN {X 0,Y 340.214,Z 342.641,A -85,B 0,C 180,E1 -15359.808,E2 -15359.808} C_VEL
LIN {X 0,Y 339.402,Z 357.789,A -85,B 0,C 180,E1 -15360.368,E2 -15360.368} C_VEL
LIN {X 0,Y 338.375,Z 371.67,A -85,B 0,C 180,E1 -15361.108,E2 -15361.108} C_VEL
LIN {X 0,Y 337.005,Z 384.862,A -85,B 0,C 180,E1 -15362.015,E2 -15362.015} C_VEL
LIN {X 0,Y 335.165,Z 398.619,A -85,B 0,C 180,E1 -15363.202,E2 -15363.202} C_VEL
LIN {X 0,Y 333.182,Z 411.194,A -85,B 0,C 180,E1 -15364.545,E2 -15364.545} C_VEL
LIN {X 0,Y 331.049,Z 422.975,A -85,B 0,C 180,E1 -15366.068,E2 -15366.068} C_VEL
LIN {X 0,Y 329.155,Z 433.572,A -85,B 0,C 180,E1 -15367.727,E2 -15367.727} C_VEL
LIN {X 0,Y 327.087,Z 443.467,A -85,B 0,C 180,E1 -15369.563,E2 -15369.563} C_VEL
LIN {X 0,Y 324.966,Z 453.119,A -85,B 0,C 180,E1 -15371.723,E2 -15371.723} C_VEL
LIN {X 0,Y 323.061,Z 462.129,A -85,B 0,C 180,E1 -15374.219,E2 -15374.219} C_VEL
LIN {X 0,Y 321.471,Z 469.386,A -85,B 0,C 180,E1 -15376.728,E2 -15376.728} C_VEL
LIN {X 0,Y 320.289,Z 475.129,A -85,B 0,C 180,E1 -15379.249,E2 -15379.249} C_VEL
LIN {X 0,Y 319.444,Z 479.701,A -85,B 0,C 180,E1 -15381.905,E2 -15381.905} C_VEL
LIN {X 0,Y 318.957,Z 481.965,A -85,B 0,C 180,E1 -15383.673,E2 -15383.673} C_VEL
LIN {X 0,Y 318.748,Z 484.222,A -85,B 0,C 180,E1 -15386.206,E2 -15386.206} C_VEL
LIN {X 0,Y 318.426,Z 485.387,A -85,B 0,C 180,E1 -15388.734,E2 -15388.734} C_VEL
LIN {X 0,Y 318.425,Z 485.4,A -85,B 0,C 180,E1 -15391.263,E2 -15391.263} C_VEL
LIN {X 0,Y 318.743,Z 484.287,A -85,B 0,C 180,E1 -15393.791,E2 -15393.791} C_VEL
LIN {X 0,Y 318.948,Z 482.085,A -85,B 0,C 180,E1 -15396.324,E2 -15396.324} C_VEL
LIN {X 0,Y 319.614,Z 478.697,A -85,B 0,C 180,E1 -15398.853,E2 -15398.853} C_VEL
LIN {X 0,Y 320.545,Z 474.05,A -85,B 0,C 180,E1 -15401.379,E2 -15401.379} C_VEL
LIN {X 0,Y 321.771,Z 468.013,A -85,B 0,C 180,E1 -15403.9,E2 -15403.9} C_VEL
LIN {X 0,Y 323.276,Z 461.473,A -85,B 0,C 180,E1 -15406.09,E2 -15406.09} C_VEL
LIN {X 0,Y 324.889,Z 453.552,A -85,B 0,C 180,E1 -15408.278,E2 -15408.278} C_VEL
LIN {X 0,Y 326.996,Z 443.994,A -85,B 0,C 180,E1 -15410.44,E2 -15410.44} C_VEL
LIN {X 0,Y 329.373,Z 432.393,A -85,B 0,C 180,E1 -15412.584,E2 -15412.584} C_VEL
LIN {X 0,Y 331.581,Z 420.562,A -85,B 0,C 180,E1 -15414.377,E2 -15414.377} C_VEL
LIN {X 0,Y 332.641,Z 414.571,A -85,B 0,C 180,E1 -15415.161,E2 -15415.161} C_VEL
LIN {X 0,Y 332.887,Z 409.908,A -85,B 0,C 180,E1 -15415.772,E2 -15415.772} C_VEL
LIN {X 0,Y 331.647,Z 402.213,A -85,B 0,C 180,E1 -15416.85,E2 -15416.85} C_VEL
LIN {X 0,Y 330.253,Z 394.339,A -85,B 0,C 180,E1 -15417.864,E2 -15417.864} C_VEL
LIN {X 0,Y 330.368,Z 389.209,A -85,B 0,C 180,E1 -15418.367,E2 -15418.367} C_VEL
LIN {X 0,Y 332.069,Z 374.614,A -85,B 0,C 180,E1 -15419.442,E2 -15419.442} C_VEL
LIN {X 0,Y 333.212,Z 360.498,A -85,B 0,C 180,E1 -15420.244,E2 -15420.244} C_VEL
LIN {X 0,Y 334.127,Z 345.467,A -85,B 0,C 180,E1 -15420.842,E2 -15420.842} C_VEL
LIN {X 0,Y 335.074,Z 317.677,A -85,B 0,C 180,E1 -15421.491,E2 -15421.491} C_VEL
LIN {X 0,Y 338.495,Z 215.506,A -85,B 0,C 180,E1 -15423.666,E2 -15423.666} C_VEL
LIN {X 0,Y 330.497,Z 198.811,A -85,B 0,C 180,E1 -15425.047,E2 -15425.047} C_VEL
LIN {X 0,Y 321.431,Z 182.214,A -85,B 0,C 180,E1 -15426.663,E2 -15426.663} C_VEL
LIN {X 0,Y 317.304,Z 175.304,A -85,B 0,C 180,E1 -15427.455,E2 -15427.455} C_VEL
LIN {X 0,Y 313.877,Z 166.5,A -85,B 0,C 180,E1 -15429.41,E2 -15429.41} C_VEL
LIN {X 0,Y 313.097,Z 165.25,A -85,B 0,C 180,E1 -15429.748,E2 -15429.748} C_VEL
LIN {X 0,Y 312.481,Z 163.155,A -85,B 0,C 180,E1 -15430.23,E2 -15430.23} C_VEL
LIN {X 0,Y 312.513,Z 163.181,A -85,B 0,C 180,E1 -15432.425,E2 -15432.425} C_VEL
LIN {X 0,Y 312.475,Z 163.188,A -85,B 0,C 180,E1 -15436.029,E2 -15436.029} C_VEL
LIN {X 0,Y 312.493,Z 163.187,A -85,B 0,C 180,E1 -15439.291,E2 -15439.291} C_VEL
LIN {X 0,Y 312.533,Z 163.177,A -85,B 0,C 180,E1 -15442.616,E2 -15442.616} C_VEL
LIN {X 0,Y 312.511,Z 163.174,A -85,B 0,C 180,E1 -15446.31,E2 -15446.31} C_VEL
LIN {X 0,Y 312.541,Z 163.16,A -85,B 0,C 180,E1 -15450.349,E2 -15450.349} C_VEL
LIN {X 0,Y 312.593,Z 163.162,A -85,B 0,C 180,E1 -15454.063,E2 -15454.063} C_VEL
LIN {X 0,Y 312.577,Z 163.175,A -85,B 0,C 180,E1 -15457.528,E2 -15457.528} C_VEL
LIN {X 0,Y 312.628,Z 163.15,A -85,B 0,C 180,E1 -15461.656,E2 -15461.656} C_VEL
LIN {X 0,Y 312.683,Z 163.15,A -85,B 0,C 180,E1 -15465.686,E2 -15465.686} C_VEL
LIN {X 0,Y 312.691,Z 163.159,A -85,B 0,C 180,E1 -15469.641,E2 -15469.641} C_VEL
LIN {X 0,Y 312.861,Z 163.123,A -85,B 0,C 180,E1 -15472.254,E2 -15472.254} C_VEL
LIN {X 0,Y 312.709,Z 163.141,A -85,B 0,C 180,E1 -15474.842,E2 -15474.842} C_VEL
LIN {X 0,Y 312.982,Z 163.109,A -85,B 0,C 180,E1 -15478.713,E2 -15478.713} C_VEL
LIN {X 0,Y 313.11,Z 163.082,A -85,B 0,C 180,E1 -15480,E2 -15480} C_VEL
LIN {X 0,Y 312.928,Z 163.125,A -85,B 0,C 180,E1 -15482.574,E2 -15482.574} C_VEL
LIN {X 0,Y 312.899,Z 163.108,A -85,B 0,C 180,E1 -15486.448,E2 -15486.448} C_VEL
LIN {X 0,Y 312.777,Z 163.143,A -85,B 0,C 180,E1 -15489.049,E2 -15489.049} C_VEL
LIN {X 0,Y 312.623,Z 163.141,A -85,B 0,C 180,E1 -15492.991,E2 -15492.991} C_VEL
LIN {X 0,Y 312.628,Z 163.162,A -85,B 0,C 180,E1 -15495.65,E2 -15495.65} C_VEL
LIN {X 0,Y 312.619,Z 163.145,A -85,B 0,C 180,E1 -15499.237,E2 -15499.237} C_VEL
LIN {X 0,Y 312.535,Z 163.172,A -85,B 0,C 180,E1 -15502.79,E2 -15502.79} C_VEL
LIN {X 0,Y 312.592,Z 163.163,A -85,B 0,C 180,E1 -15505.936,E2 -15505.936} C_VEL
LIN {X 0,Y 312.528,Z 163.164,A -85,B 0,C 180,E1 -15509.652,E2 -15509.652} C_VEL
LIN {X 0,Y 312.51,Z 163.171,A -85,B 0,C 180,E1 -15513.69,E2 -15513.69} C_VEL
LIN {X 0,Y 312.529,Z 163.173,A -85,B 0,C 180,E1 -15517.384,E2 -15517.384} C_VEL
LIN {X 0,Y 312.481,Z 163.137,A -85,B 0,C 180,E1 -15520.71,E2 -15520.71} C_VEL
LIN {X 0,Y 312.511,Z 163.183,A -85,B 0,C 180,E1 -15524.199,E2 -15524.199} C_VEL
LIN {X 0,Y 312.555,Z 163.316,A -85,B 0,C 180,E1 -15526.074,E2 -15526.074} C_VEL
LIN {X 0,Y 318.003,Z 181.951,A -85,B 0,C 180,E1 -15529.978,E2 -15529.978} C_VEL
LIN {X 0,Y 320.956,Z 192.181,A -85,B 0,C 180,E1 -15531.964,E2 -15531.964} C_VEL
LIN {X 0,Y 329.12,Z 213.377,A -85,B 0,C 180,E1 -15534.237,E2 -15534.237} C_VEL
LIN {X 0,Y 331.145,Z 231.369,A -85,B 0,C 180,E1 -15534.994,E2 -15534.994} C_VEL
LIN {X 0,Y 335.965,Z 277.612,A -85,B 0,C 180,E1 -15536.715,E2 -15536.715} C_VEL
LIN {X 0,Y 332.406,Z 387.611,A -85,B 0,C 180,E1 -15539.069,E2 -15539.069} C_VEL
LIN {X 0,Y 331.355,Z 403.512,A -85,B 0,C 180,E1 -15539.579,E2 -15539.579} C_VEL
LIN {X 0,Y 329.678,Z 418.631,A -85,B 0,C 180,E1 -15540.29,E2 -15540.29} C_VEL
LIN {X 0,Y 327.866,Z 432.251,A -85,B 0,C 180,E1 -15541.166,E2 -15541.166} C_VEL
LIN {X 0,Y 325.718,Z 445.648,A -85,B 0,C 180,E1 -15542.263,E2 -15542.263} C_VEL
LIN {X 0,Y 323.507,Z 458.314,A -85,B 0,C 180,E1 -15543.556,E2 -15543.556} C_VEL
LIN {X 0,Y 321.057,Z 470.575,A -85,B 0,C 180,E1 -15545.08,E2 -15545.08} C_VEL
LIN {X 0,Y 318.655,Z 482.822,A -85,B 0,C 180,E1 -15546.955,E2 -15546.955} C_VEL
LIN {X 0,Y 316.598,Z 492.857,A -85,B 0,C 180,E1 -15548.802,E2 -15548.802} C_VEL
LIN {X 0,Y 314.661,Z 503.204,A -85,B 0,C 180,E1 -15551.105,E2 -15551.105} C_VEL
LIN {X 0,Y 313.052,Z 511.581,A -85,B 0,C 180,E1 -15553.369,E2 -15553.369} C_VEL
LIN {X 0,Y 312.057,Z 518.551,A -85,B 0,C 180,E1 -15555.658,E2 -15555.658} C_VEL
LIN {X 0,Y 311.286,Z 525.026,A -85,B 0,C 180,E1 -15558.278,E2 -15558.278} C_VEL
LIN {X 0,Y 311.028,Z 530.056,A -85,B 0,C 180,E1 -15560.901,E2 -15560.901} C_VEL
LIN {X 0,Y 311.164,Z 533.87,A -85,B 0,C 180,E1 -15563.61,E2 -15563.61} C_VEL
LIN {X 0,Y 311.203,Z 536.197,A -85,B 0,C 180,E1 -15566.117,E2 -15566.117} C_VEL
LIN {X 0,Y 311.388,Z 536.972,A -85,B 0,C 180,E1 -15567.414,E2 -15567.414} C_VEL
LIN {X 0,Y 311.547,Z 537.605,A -85,B 0,C 180,E1 -15570.002,E2 -15570.002} C_VEL
LIN {X 0,Y 311.389,Z 536.967,A -85,B 0,C 180,E1 -15572.589,E2 -15572.589} C_VEL
LIN {X 0,Y 311.214,Z 535.123,A -85,B 0,C 180,E1 -15575.184,E2 -15575.184} C_VEL
LIN {X 0,Y 311.222,Z 533.748,A -85,B 0,C 180,E1 -15576.485,E2 -15576.485} C_VEL
LIN {X 0,Y 311.063,Z 530.022,A -85,B 0,C 180,E1 -15579.101,E2 -15579.101} C_VEL
LIN {X 0,Y 311.322,Z 524.977,A -85,B 0,C 180,E1 -15581.724,E2 -15581.724} C_VEL
LIN {X 0,Y 312.065,Z 518.217,A -85,B 0,C 180,E1 -15584.443,E2 -15584.443} C_VEL
LIN {X 0,Y 313.261,Z 510.371,A -85,B 0,C 180,E1 -15586.959,E2 -15586.959} C_VEL
LIN {X 0,Y 314.916,Z 501.743,A -85,B 0,C 180,E1 -15589.22,E2 -15589.22} C_VEL
LIN {X 0,Y 316.588,Z 492.78,A -85,B 0,C 180,E1 -15591.194,E2 -15591.194} C_VEL
LIN {X 0,Y 318.614,Z 482.685,A -85,B 0,C 180,E1 -15593.051,E2 -15593.051} C_VEL
LIN {X 0,Y 321.099,Z 470.405,A -85,B 0,C 180,E1 -15594.92,E2 -15594.92} C_VEL
LIN {X 0,Y 323.509,Z 458.113,A -85,B 0,C 180,E1 -15596.447,E2 -15596.447} C_VEL
LIN {X 0,Y 325.166,Z 450.384,A -85,B 0,C 180,E1 -15597.364,E2 -15597.364} C_VEL
LIN {X 0,Y 328.266,Z 437.895,A -85,B 0,C 180,E1 -15598.799,E2 -15598.799} C_VEL
LIN {X 0,Y 331.428,Z 424.31,A -85,B 0,C 180,E1 -15600.066,E2 -15600.066} C_VEL
LIN {X 0,Y 334.605,Z 409.754,A -85,B 0,C 180,E1 -15601.147,E2 -15601.147} C_VEL
LIN {X 0,Y 337.539,Z 393.754,A -85,B 0,C 180,E1 -15602.071,E2 -15602.071} C_VEL
LIN {X 0,Y 340.008,Z 375.912,A -85,B 0,C 180,E1 -15602.818,E2 -15602.818} C_VEL
LIN {X 0,Y 347.054,Z 313.514,A -85,B 0,C 180,E1 -15604.998,E2 -15604.998} C_VEL
LIN {X 0,Y 351.221,Z 280.381,A -85,B 0,C 180,E1 -15606.212,E2 -15606.212} C_VEL
LIN {X 0,Y 351.637,Z 267.076,A -85,B 0,C 180,E1 -15607.076,E2 -15607.076} C_VEL
LIN {X 0,Y 351.567,Z 253.546,A -85,B 0,C 180,E1 -15608.198,E2 -15608.198} C_VEL
LIN {X 0,Y 351.37,Z 242.922,A -85,B 0,C 180,E1 -15609.243,E2 -15609.243} C_VEL
LIN {X 0,Y 349.331,Z 238.432,A -85,B 0,C 180,E1 -15610.53,E2 -15610.53} C_VEL
LIN {X 0,Y 346.573,Z 232.921,A -85,B 0,C 180,E1 -15612.715,E2 -15612.715} C_VEL
LIN {X 0,Y 345.062,Z 230.559,A -85,B 0,C 180,E1 -15614.316,E2 -15614.316} C_VEL
LIN {X 0,Y 343.863,Z 228.465,A -85,B 0,C 180,E1 -15616.597,E2 -15616.597} C_VEL
LIN {X 0,Y 343.663,Z 228.069,A -85,B 0,C 180,E1 -15617.557,E2 -15617.557} C_VEL
LIN {X 0,Y 344.041,Z 228.149,A -85,B 0,C 180,E1 -15619.949,E2 -15619.949} C_VEL
LIN {X 0,Y 345.407,Z 230.76,A -85,B 0,C 180,E1 -15622.381,E2 -15622.381} C_VEL
LIN {X 0,Y 346.803,Z 232.791,A -85,B 0,C 180,E1 -15623.778,E2 -15623.778} C_VEL
LIN {X 0,Y 349.224,Z 237.131,A -85,B 0,C 180,E1 -15625.703,E2 -15625.703} C_VEL
LIN {X 0,Y 351.394,Z 241.728,A -85,B 0,C 180,E1 -15627.143,E2 -15627.143} C_VEL
LIN {X 0,Y 353.365,Z 246.264,A -85,B 0,C 180,E1 -15628.303,E2 -15628.303} C_VEL
LIN {X 0,Y 354.095,Z 253.874,A -85,B 0,C 180,E1 -15629.239,E2 -15629.239} C_VEL
LIN {X 0,Y 342.24,Z 330.973,A -85,B 0,C 180,E1 -15632.557,E2 -15632.557} C_VEL
LIN {X 0,Y 340.324,Z 347.057,A -85,B 0,C 180,E1 -15633.393,E2 -15633.393} C_VEL
LIN {X 0,Y 338.397,Z 360.547,A -85,B 0,C 180,E1 -15634.308,E2 -15634.308} C_VEL
LIN {X 0,Y 335.786,Z 375.193,A -85,B 0,C 180,E1 -15635.584,E2 -15635.584} C_VEL
LIN {X 0,Y 333.361,Z 387.031,A -85,B 0,C 180,E1 -15636.88,E2 -15636.88} C_VEL
LIN {X 0,Y 331.056,Z 396.927,A -85,B 0,C 180,E1 -15638.191,E2 -15638.191} C_VEL
LIN {X 0,Y 328.235,Z 407.889,A -85,B 0,C 180,E1 -15639.966,E2 -15639.966} C_VEL
LIN {X 0,Y 325.872,Z 416.563,A -85,B 0,C 180,E1 -15641.712,E2 -15641.712} C_VEL
LIN {X 0,Y 323.009,Z 425.312,A -85,B 0,C 180,E1 -15643.894,E2 -15643.894} C_VEL
LIN {X 0,Y 320.702,Z 431.965,A -85,B 0,C 180,E1 -15646.051,E2 -15646.051} C_VEL
LIN {X 0,Y 318.842,Z 436.424,A -85,B 0,C 180,E1 -15647.913,E2 -15647.913} C_VEL
LIN {X 0,Y 317.387,Z 439.761,A -85,B 0,C 180,E1 -15649.797,E2 -15649.797} C_VEL
LIN {X 0,Y 316.425,Z 441.45,A -85,B 0,C 180,E1 -15651.056,E2 -15651.056} C_VEL
LIN {X 0,Y 315.644,Z 442.681,A -85,B 0,C 180,E1 -15652.323,E2 -15652.323} C_VEL
LIN {X 0,Y 314.534,Z 443.894,A -85,B 0,C 180,E1 -15654.872,E2 -15654.872} C_VEL
LIN {X 0,Y 313.989,Z 443.904,A -85,B 0,C 180,E1 -15656.15,E2 -15656.15} C_VEL
LIN {X 0,Y 313.614,Z 443.448,A -85,B 0,C 180,E1 -15657.431,E2 -15657.431} C_VEL
LIN {X 0,Y 313.214,Z 442.601,A -85,B 0,C 180,E1 -15658.714,E2 -15658.714} C_VEL
LIN {X 0,Y 312.89,Z 441.345,A -85,B 0,C 180,E1 -15660,E2 -15660} C_VEL
LIN {X 0,Y 312.769,Z 438.607,A -85,B 0,C 180,E1 -15661.932,E2 -15661.932} C_VEL
LIN {X 0,Y 312.624,Z 434.877,A -85,B 0,C 180,E1 -15663.867,E2 -15663.867} C_VEL
LIN {X 0,Y 312.797,Z 430.045,A -85,B 0,C 180,E1 -15665.803,E2 -15665.803} C_VEL
LIN {X 0,Y 313.074,Z 424.014,A -85,B 0,C 180,E1 -15667.741,E2 -15667.741} C_VEL
LIN {X 0,Y 313.43,Z 416.875,A -85,B 0,C 180,E1 -15669.617,E2 -15669.617} C_VEL
LIN {X 0,Y 314.054,Z 407.535,A -85,B 0,C 180,E1 -15671.619,E2 -15671.619} C_VEL
LIN {X 0,Y 314.793,Z 396.435,A -85,B 0,C 180,E1 -15673.558,E2 -15673.558} C_VEL
LIN {X 0,Y 315.54,Z 385.042,A -85,B 0,C 180,E1 -15675.172,E2 -15675.172} C_VEL
LIN {X 0,Y 316.364,Z 372.523,A -85,B 0,C 180,E1 -15676.62,E2 -15676.62} C_VEL
LIN {X 0,Y 317.068,Z 359.136,A -85,B 0,C 180,E1 -15677.862,E2 -15677.862} C_VEL
LIN {X 0,Y 317.773,Z 345.149,A -85,B 0,C 180,E1 -15678.872,E2 -15678.872} C_VEL
LIN {X 0,Y 318.225,Z 330.928,A -85,B 0,C 180,E1 -15679.64,E2 -15679.64} C_VEL
LIN {X 0,Y 318.879,Z 307.578,A -85,B 0,C 180,E1 -15680.48,E2 -15680.48} C_VEL
LIN {X 0,Y 321.805,Z 231.11,A -85,B 0,C 180,E1 -15682.986,E2 -15682.986} C_VEL
LIN {X 0,Y 318.158,Z 204.643,A -85,B 0,C 180,E1 -15684.121,E2 -15684.121} C_VEL
LIN {X 0,Y 319.284,Z 194.076,A -85,B 0,C 180,E1 -15686.471,E2 -15686.471} C_VEL
LIN {X 0,Y 317.531,Z 184.645,A -85,B 0,C 180,E1 -15688.802,E2 -15688.802} C_VEL
LIN {X 0,Y 313.899,Z 169.023,A -85,B 0,C 180,E1 -15692.862,E2 -15692.862} C_VEL
LIN {X 0,Y 312.55,Z 163.178,A -85,B 0,C 180,E1 -15694.449,E2 -15694.449} C_VEL
LIN {X 0,Y 312.492,Z 163.185,A -85,B 0,C 180,E1 -15698.078,E2 -15698.078} C_VEL
LIN {X 0,Y 312.494,Z 163.174,A -85,B 0,C 180,E1 -15700.709,E2 -15700.709} C_VEL
LIN {X 0,Y 312.478,Z 163.176,A -85,B 0,C 180,E1 -15704.205,E2 -15704.205} C_VEL
LIN {X 0,Y 312.492,Z 163.181,A -85,B 0,C 180,E1 -15707.917,E2 -15707.917} C_VEL
LIN {X 0,Y 312.525,Z 163.255,A -85,B 0,C 180,E1 -15709.959,E2 -15709.959} C_VEL
LIN {X 0,Y 314.233,Z 167.821,A -85,B 0,C 180,E1 -15711.002,E2 -15711.002} C_VEL
LIN {X 0,Y 317.561,Z 175.724,A -85,B 0,C 180,E1 -15712.75,E2 -15712.75} C_VEL
LIN {X 0,Y 325.712,Z 189.792,A -85,B 0,C 180,E1 -15714.23,E2 -15714.23} C_VEL
LIN {X 0,Y 334.537,Z 206.994,A -85,B 0,C 180,E1 -15715.773,E2 -15715.773} C_VEL
LIN {X 0,Y 338.418,Z 215.339,A -85,B 0,C 180,E1 -15716.438,E2 -15716.438} C_VEL
LIN {X 0,Y 335.059,Z 316.433,A -85,B 0,C 180,E1 -15718.592,E2 -15718.592} C_VEL
LIN {X 0,Y 334.066,Z 344.531,A -85,B 0,C 180,E1 -15719.236,E2 -15719.236} C_VEL
LIN {X 0,Y 333.108,Z 360.512,A -85,B 0,C 180,E1 -15719.862,E2 -15719.862} C_VEL
LIN {X 0,Y 331.954,Z 374.917,A -85,B 0,C 180,E1 -15720.683,E2 -15720.683} C_VEL
LIN {X 0,Y 330.362,Z 389.249,A -85,B 0,C 180,E1 -15721.747,E2 -15721.747} C_VEL
LIN {X 0,Y 328.454,Z 402.244,A -85,B 0,C 180,E1 -15722.953,E2 -15722.953} C_VEL
LIN {X 0,Y 326.104,Z 415.525,A -85,B 0,C 180,E1 -15724.466,E2 -15724.466} C_VEL
LIN {X 0,Y 323.652,Z 428.533,A -85,B 0,C 180,E1 -15726.313,E2 -15726.313} C_VEL
LIN {X 0,Y 321.532,Z 439.315,A -85,B 0,C 180,E1 -15728.185,E2 -15728.185} C_VEL
LIN {X 0,Y 319.177,Z 449.77,A -85,B 0,C 180,E1 -15730.378,E2 -15730.378} C_VEL
LIN {X 0,Y 317.289,Z 457.995,A -85,B 0,C 180,E1 -15732.464,E2 -15732.464} C_VEL
LIN {X 0,Y 315.714,Z 464.669,A -85,B 0,C 180,E1 -15734.505,E2 -15734.505} C_VEL
LIN {X 0,Y 314.245,Z 471.524,A -85,B 0,C 180,E1 -15737.075,E2 -15737.075} C_VEL
LIN {X 0,Y 313.069,Z 476.91,A -85,B 0,C 180,E1 -15739.653,E2 -15739.653} C_VEL
LIN {X 0,Y 312.272,Z 480.974,A -85,B 0,C 180,E1 -15742.238,E2 -15742.238} C_VEL
LIN {X 0,Y 311.854,Z 483.815,A -85,B 0,C 180,E1 -15744.826,E2 -15744.826} C_VEL
LIN {X 0,Y 311.491,Z 485.527,A -85,B 0,C 180,E1 -15747.412,E2 -15747.412} C_VEL
LIN {X 0,Y 311.329,Z 486.124,A -85,B 0,C 180,E1 -15749.998,E2 -15749.998} C_VEL
LIN {X 0,Y 311.49,Z 485.565,A -85,B 0,C 180,E1 -15752.585,E2 -15752.585} C_VEL
LIN {X 0,Y 311.817,Z 483.908,A -85,B 0,C 180,E1 -15755.171,E2 -15755.171} C_VEL
LIN {X 0,Y 312.289,Z 481.121,A -85,B 0,C 180,E1 -15757.759,E2 -15757.759} C_VEL
LIN {X 0,Y 313.042,Z 477.125,A -85,B 0,C 180,E1 -15760.345,E2 -15760.345} C_VEL
LIN {X 0,Y 314.188,Z 471.8,A -85,B 0,C 180,E1 -15762.924,E2 -15762.924} C_VEL
LIN {X 0,Y 315.675,Z 465.003,A -85,B 0,C 180,E1 -15765.494,E2 -15765.494} C_VEL
LIN {X 0,Y 317.066,Z 458.837,A -85,B 0,C 180,E1 -15767.408,E2 -15767.408} C_VEL
LIN {X 0,Y 319.087,Z 450.228,A -85,B 0,C 180,E1 -15769.625,E2 -15769.625} C_VEL
LIN {X 0,Y 321.058,Z 441.444,A -85,B 0,C 180,E1 -15771.508,E2 -15771.508} C_VEL
LIN {X 0,Y 323.223,Z 431.077,A -85,B 0,C 180,E1 -15773.377,E2 -15773.377} C_VEL
LIN {X 0,Y 325.382,Z 419.772,A -85,B 0,C 180,E1 -15775.078,E2 -15775.078} C_VEL
LIN {X 0,Y 327.641,Z 407.418,A -85,B 0,C 180,E1 -15776.599,E2 -15776.599} C_VEL
LIN {X 0,Y 329.715,Z 393.852,A -85,B 0,C 180,E1 -15777.963,E2 -15777.963} C_VEL
LIN {X 0,Y 330.368,Z 389.209,A -85,B 0,C 180,E1 -15778.367,E2 -15778.367} C_VEL
LIN {X 0,Y 330.48,Z 383.975,A -85,B 0,C 180,E1 -15778.843,E2 -15778.843} C_VEL
LIN {X 0,Y 328.915,Z 375.525,A -85,B 0,C 180,E1 -15779.707,E2 -15779.707} C_VEL
LIN {X 0,Y 327.23,Z 366.879,A -85,B 0,C 180,E1 -15780.499,E2 -15780.499} C_VEL
LIN {X 0,Y 327.098,Z 361.342,A -85,B 0,C 180,E1 -15780.853,E2 -15780.853} C_VEL
LIN {X 0,Y 328.089,Z 345.962,A -85,B 0,C 180,E1 -15781.474,E2 -15781.474} C_VEL
LIN {X 0,Y 328.99,Z 319.906,A -85,B 0,C 180,E1 -15782.097,E2 -15782.097} C_VEL
LIN {X 0,Y 332.608,Z 217.71,A -85,B 0,C 180,E1 -15784.298,E2 -15784.298} C_VEL
LIN {X 0,Y 324.049,Z 200.002,A -85,B 0,C 180,E1 -15785.831,E2 -15785.831} C_VEL
LIN {X 0,Y 314.993,Z 183.709,A -85,B 0,C 180,E1 -15787.511,E2 -15787.511} C_VEL
LIN {X 0,Y 310.255,Z 175.907,A -85,B 0,C 180,E1 -15788.468,E2 -15788.468} C_VEL
LIN {X 0,Y 306.675,Z 167.244,A -85,B 0,C 180,E1 -15790.487,E2 -15790.487} C_VEL
LIN {X 0,Y 305.43,Z 164.04,A -85,B 0,C 180,E1 -15791.279,E2 -15791.279} C_VEL
LIN {X 0,Y 305.407,Z 164.059,A -85,B 0,C 180,E1 -15794.49,E2 -15794.49} C_VEL
LIN {X 0,Y 305.468,Z 164.052,A -85,B 0,C 180,E1 -15798.148,E2 -15798.148} C_VEL
LIN {X 0,Y 305.5,Z 164.045,A -85,B 0,C 180,E1 -15801.601,E2 -15801.601} C_VEL
LIN {X 0,Y 305.454,Z 164.049,A -85,B 0,C 180,E1 -15804.886,E2 -15804.886} C_VEL
LIN {X 0,Y 305.448,Z 164.061,A -85,B 0,C 180,E1 -15808.352,E2 -15808.352} C_VEL
LIN {X 0,Y 305.52,Z 164.04,A -85,B 0,C 180,E1 -15811.114,E2 -15811.114} C_VEL
LIN {X 0,Y 305.563,Z 164.037,A -85,B 0,C 180,E1 -15814.087,E2 -15814.087} C_VEL
LIN {X 0,Y 305.49,Z 164.058,A -85,B 0,C 180,E1 -15818.402,E2 -15818.402} C_VEL
LIN {X 0,Y 305.58,Z 164.025,A -85,B 0,C 180,E1 -15821.217,E2 -15821.217} C_VEL
LIN {X 0,Y 305.638,Z 164.03,A -85,B 0,C 180,E1 -15825.348,E2 -15825.348} C_VEL
LIN {X 0,Y 305.628,Z 164.038,A -85,B 0,C 180,E1 -15829.399,E2 -15829.399} C_VEL
